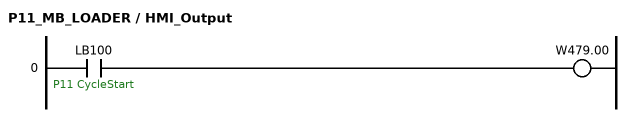
; [picture p120: P11_MB_LOADER / HMI_Output, rungs 0-0]
; rung 0
LD LB100  ; P11 CycleStart
OUT W479.00

### Section Autorun

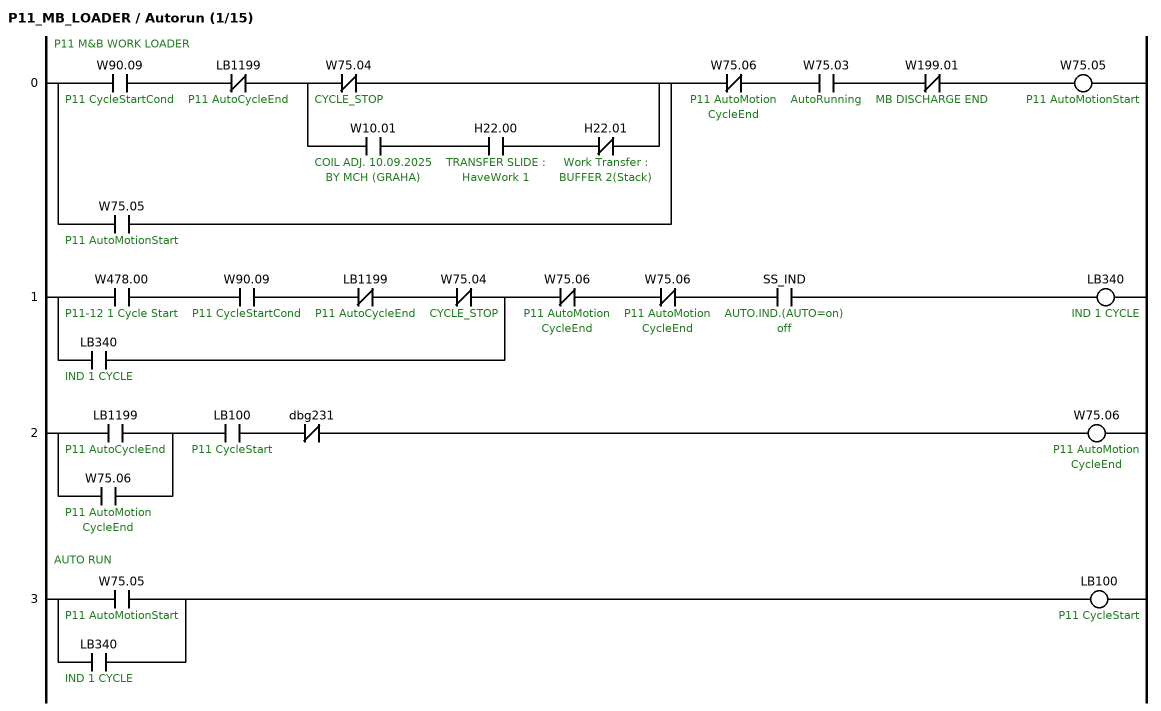
; rung 0: P11 M&B WORK LOADER
LD W90.09  ; P11 CycleStartCond
ANDNOT LB1199  ; P11 AutoCycleEnd
LDNOT W75.04  ; CYCLE_STOP
LD W10.01  ; COIL ADJ. 10.09.2025 BY MCH (GRAHA)
AND H22.00  ; TRANSFER SLIDE : HaveWork 1
ANDNOT H22.01  ; Work Transfer : BUFFER 2(Stack)
ORLD
ANDLD
OR W75.05  ; P11 AutoMotionStart
ANDNOT W75.06  ; P11 AutoMotion CycleEnd
AND W75.03  ; AutoRunning
ANDNOT W199.01  ; MB DISCHARGE END
OUT W75.05  ; P11 AutoMotionStart
; rung 1
LD W478.00  ; P11-12 1 Cycle Start
AND W90.09  ; P11 CycleStartCond
ANDNOT LB1199  ; P11 AutoCycleEnd
ANDNOT W75.04  ; CYCLE_STOP
OR LB340  ; IND 1 CYCLE
ANDNOT W75.06  ; P11 AutoMotion CycleEnd
ANDNOT W75.06  ; P11 AutoMotion CycleEnd
AND SS_IND  ; AUTO.IND.(AUTO=on) off
OUT LB340  ; IND 1 CYCLE
; rung 2
LD LB1199  ; P11 AutoCycleEnd
OR W75.06  ; P11 AutoMotion CycleEnd
AND LB100  ; P11 CycleStart
ANDNOT dbg231
OUT W75.06  ; P11 AutoMotion CycleEnd
; rung 3: AUTO RUN
LD W75.05  ; P11 AutoMotionStart
OR LB340  ; IND 1 CYCLE
OUT LB100  ; P11 CycleStart

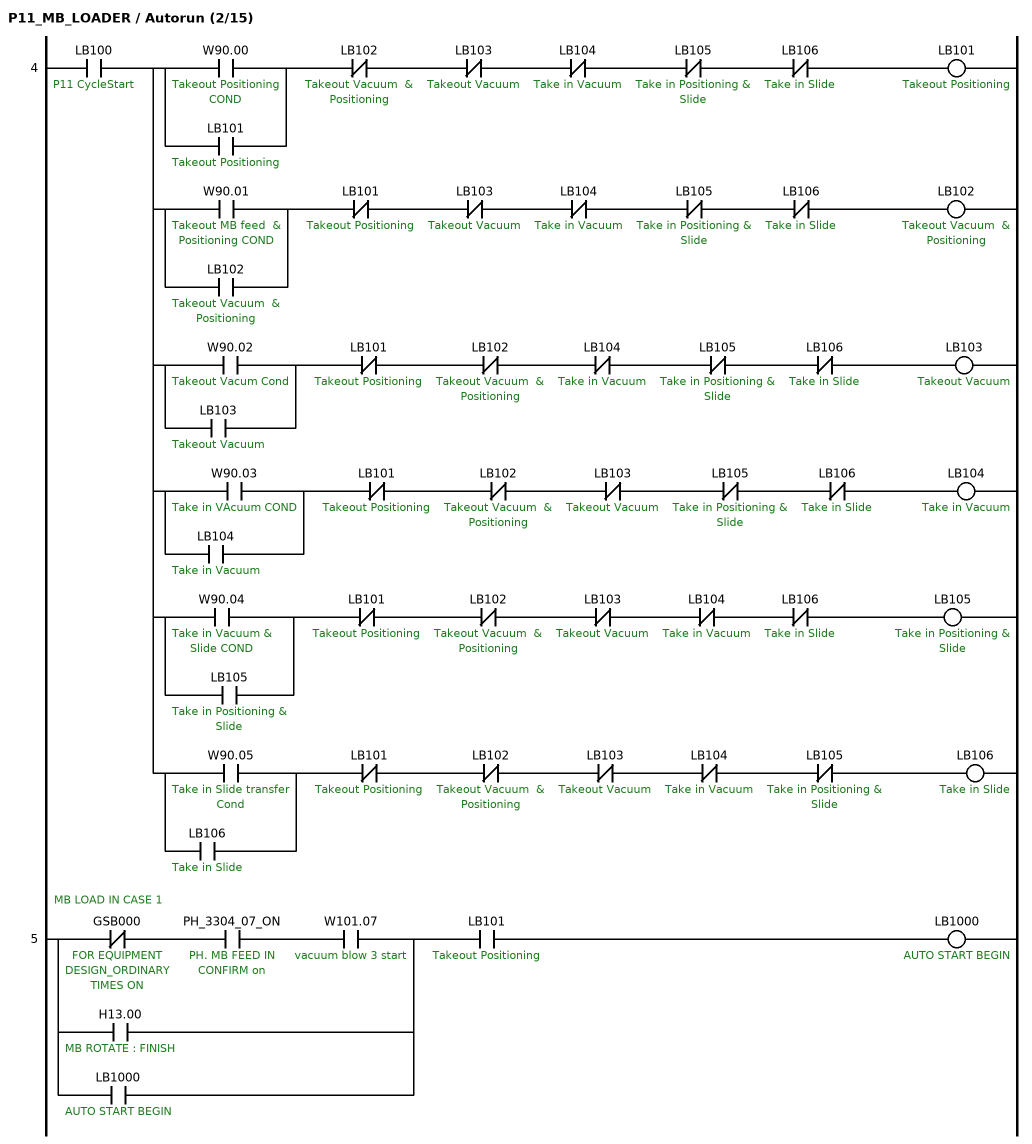
; rung 4
LD LB100  ; P11 CycleStart
OUT TR0
LD W90.00  ; Takeout Positioning COND
OR LB101  ; Takeout Positioning
ANDLD
ANDNOT LB102  ; Takeout Vacuum  & Positioning
ANDNOT LB103  ; Takeout Vacuum
ANDNOT LB104  ; Take in Vacuum
ANDNOT LB105  ; Take in Positioning & Slide
ANDNOT LB106  ; Take in Slide
OUT LB101  ; Takeout Positioning
LD TR0
LD W90.01  ; Takeout MB feed  & Positioning COND
OR LB102  ; Takeout Vacuum  & Positioning
ANDLD
ANDNOT LB101  ; Takeout Positioning
ANDNOT LB103  ; Takeout Vacuum
ANDNOT LB104  ; Take in Vacuum
ANDNOT LB105  ; Take in Positioning & Slide
ANDNOT LB106  ; Take in Slide
OUT LB102  ; Takeout Vacuum  & Positioning
LD TR0
LD W90.02  ; Takeout Vacum Cond
OR LB103  ; Takeout Vacuum
ANDLD
ANDNOT LB101  ; Takeout Positioning
ANDNOT LB102  ; Takeout Vacuum  & Positioning
ANDNOT LB104  ; Take in Vacuum
ANDNOT LB105  ; Take in Positioning & Slide
ANDNOT LB106  ; Take in Slide
OUT LB103  ; Takeout Vacuum
LD TR0
LD W90.03  ; Take in VAcuum COND
OR LB104  ; Take in Vacuum
ANDLD
ANDNOT LB101  ; Takeout Positioning
ANDNOT LB102  ; Takeout Vacuum  & Positioning
ANDNOT LB103  ; Takeout Vacuum
ANDNOT LB105  ; Take in Positioning & Slide
ANDNOT LB106  ; Take in Slide
OUT LB104  ; Take in Vacuum
LD TR0
LD W90.04  ; Take in Vacuum & Slide COND
OR LB105  ; Take in Positioning & Slide
ANDLD
ANDNOT LB101  ; Takeout Positioning
ANDNOT LB102  ; Takeout Vacuum  & Positioning
ANDNOT LB103  ; Takeout Vacuum
ANDNOT LB104  ; Take in Vacuum
ANDNOT LB106  ; Take in Slide
OUT LB105  ; Take in Positioning & Slide
LD TR0
LD W90.05  ; Take in Slide transfer Cond
OR LB106  ; Take in Slide
ANDLD
ANDNOT LB101  ; Takeout Positioning
ANDNOT LB102  ; Takeout Vacuum  & Positioning
ANDNOT LB103  ; Takeout Vacuum
ANDNOT LB104  ; Take in Vacuum
ANDNOT LB105  ; Take in Positioning & Slide
OUT LB106  ; Take in Slide
; rung 5: MB LOAD IN CASE 1
LDNOT GSB000  ; FOR EQUIPMENT DESIGN_ORDINARY TIMES ON
AND PH_3304_07_ON  ; PH. MB FEED IN CONFIRM on
AND W101.07  ; vacuum blow 3 start
OR H13.00  ; MB ROTATE : FINISH
OR LB1000  ; AUTO START BEGIN
AND LB101  ; Takeout Positioning
OUT LB1000  ; AUTO START BEGIN

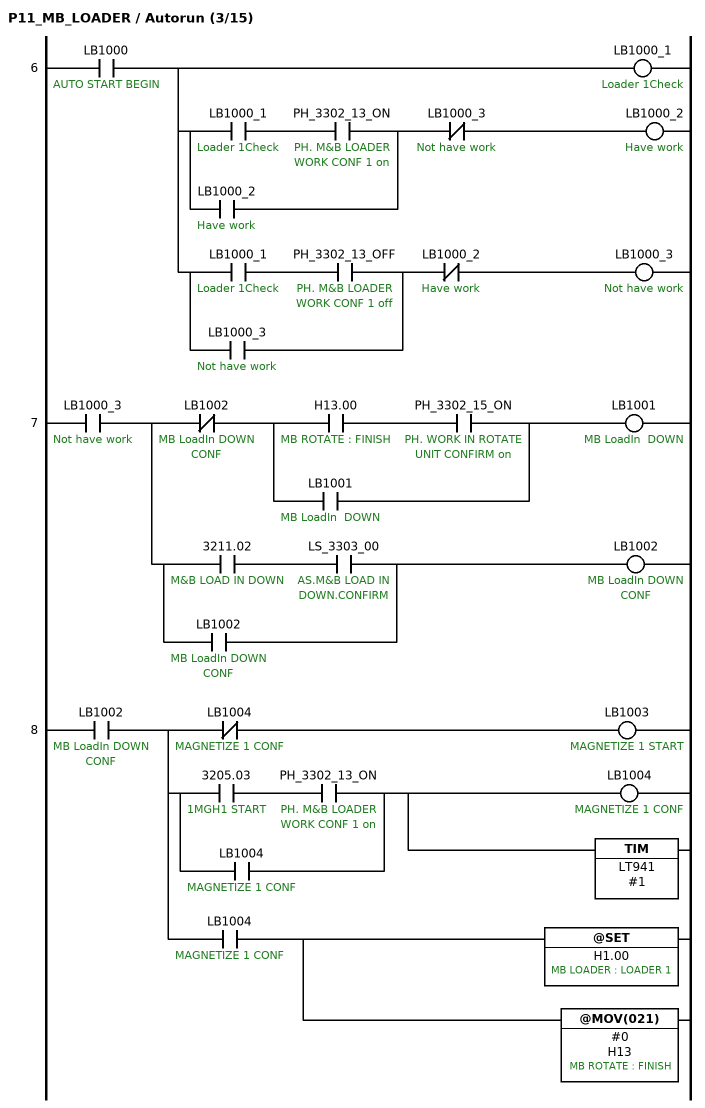
; rung 6
LD LB1000  ; AUTO START BEGIN
OUT TR0
OUT LB1000_1  ; Loader 1Check
LD LB1000_1  ; Loader 1Check
AND PH_3302_13_ON  ; PH. M&B LOADER WORK CONF 1 on
OR LB1000_2  ; Have work
ANDLD
ANDNOT LB1000_3  ; Not have work
OUT LB1000_2  ; Have work
LD TR0
LD LB1000_1  ; Loader 1Check
AND PH_3302_13_OFF  ; PH. M&B LOADER WORK CONF 1 off
OR LB1000_3  ; Not have work
ANDLD
ANDNOT LB1000_2  ; Have work
OUT LB1000_3  ; Not have work
; rung 7
LD LB1000_3  ; Not have work
OUT TR0
ANDNOT LB1002  ; MB LoadIn DOWN CONF
LD H13.00  ; MB ROTATE : FINISH
AND PH_3302_15_ON  ; PH. WORK IN ROTATE UNIT CONFIRM on
OR LB1001  ; MB LoadIn  DOWN
ANDLD
OUT LB1001  ; MB LoadIn  DOWN
LD TR0
LD 3211.02  ; M&B LOAD IN DOWN
AND LS_3303_00  ; AS.M&B LOAD IN DOWN.CONFIRM
OR LB1002  ; MB LoadIn DOWN CONF
ANDLD
OUT LB1002  ; MB LoadIn DOWN CONF
; rung 8
LD LB1002  ; MB LoadIn DOWN CONF
OUT TR0
ANDNOT LB1004  ; MAGNETIZE 1 CONF
OUT LB1003  ; MAGNETIZE 1 START
LD TR0
LD 3205.03  ; 1MGH1 START
AND PH_3302_13_ON  ; PH. M&B LOADER WORK CONF 1 on
OR LB1004  ; MAGNETIZE 1 CONF
ANDLD
OUT LB1004  ; MAGNETIZE 1 CONF
TIM LT941 #1
LD TR0
AND LB1004  ; MAGNETIZE 1 CONF
@SET H1.00  ; MB LOADER : LOADER 1
@MOV(021) #0 H13  ; MB ROTATE : FINISH

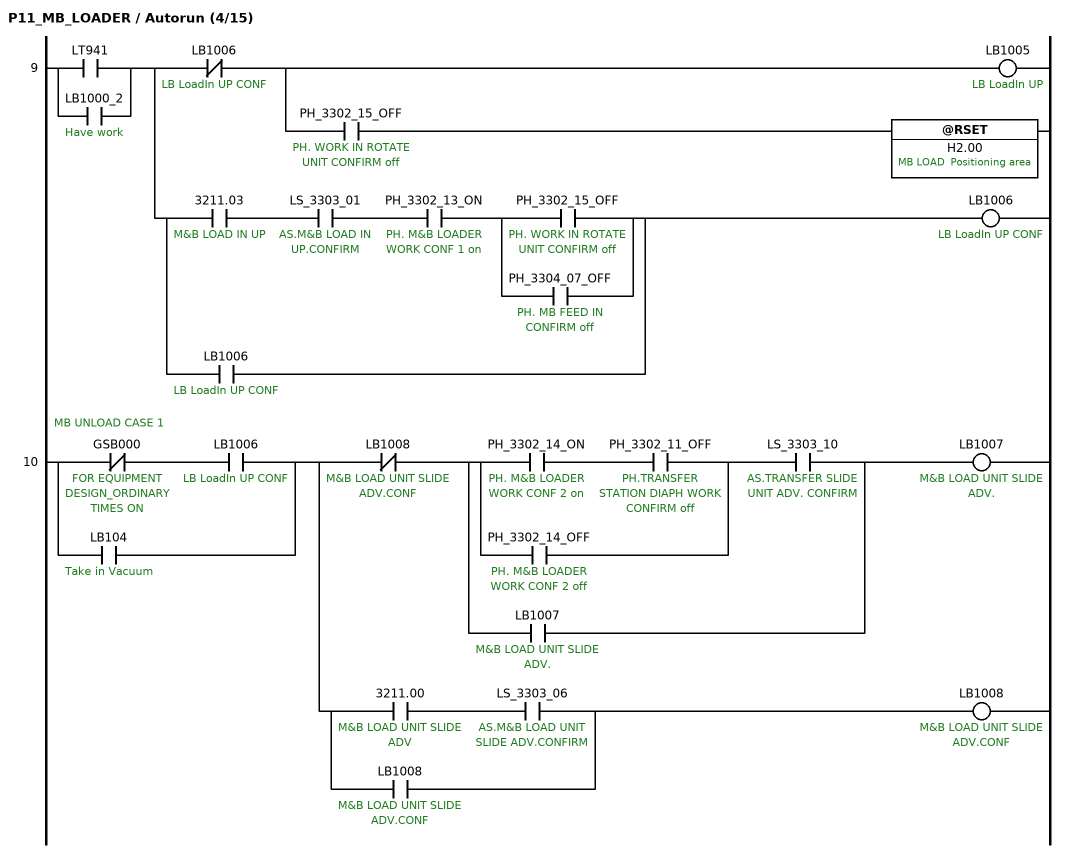
; rung 9
LD LT941
OR LB1000_2  ; Have work
OUT TR0
ANDNOT LB1006  ; LB LoadIn UP CONF
OUT LB1005  ; LB LoadIn UP
AND PH_3302_15_OFF  ; PH. WORK IN ROTATE UNIT CONFIRM off
@RSET H2.00  ; MB LOAD  Positioning area
LD TR0
LD 3211.03  ; M&B LOAD IN UP
AND LS_3303_01  ; AS.M&B LOAD IN UP.CONFIRM
AND PH_3302_13_ON  ; PH. M&B LOADER WORK CONF 1 on
LD PH_3302_15_OFF  ; PH. WORK IN ROTATE UNIT CONFIRM off
OR PH_3304_07_OFF  ; PH. MB FEED IN CONFIRM off
ANDLD
OR LB1006  ; LB LoadIn UP CONF
ANDLD
OUT LB1006  ; LB LoadIn UP CONF
; rung 10: MB UNLOAD CASE 1
LDNOT GSB000  ; FOR EQUIPMENT DESIGN_ORDINARY TIMES ON
AND LB1006  ; LB LoadIn UP CONF
OR LB104  ; Take in Vacuum
OUT TR0
ANDNOT LB1008  ; M&B LOAD UNIT SLIDE ADV.CONF
LD PH_3302_14_ON  ; PH. M&B LOADER WORK CONF 2 on
AND PH_3302_11_OFF  ; PH.TRANSFER STATION DIAPH WORK CONFIRM off
OR PH_3302_14_OFF  ; PH. M&B LOADER WORK CONF 2 off
AND LS_3303_10  ; AS.TRANSFER SLIDE UNIT ADV. CONFIRM
OR LB1007  ; M&B LOAD UNIT SLIDE ADV.
ANDLD
OUT LB1007  ; M&B LOAD UNIT SLIDE ADV.
LD TR0
LD 3211.00  ; M&B LOAD UNIT SLIDE ADV
AND LS_3303_06  ; AS.M&B LOAD UNIT SLIDE ADV.CONFIRM
OR LB1008  ; M&B LOAD UNIT SLIDE ADV.CONF
ANDLD
OUT LB1008  ; M&B LOAD UNIT SLIDE ADV.CONF

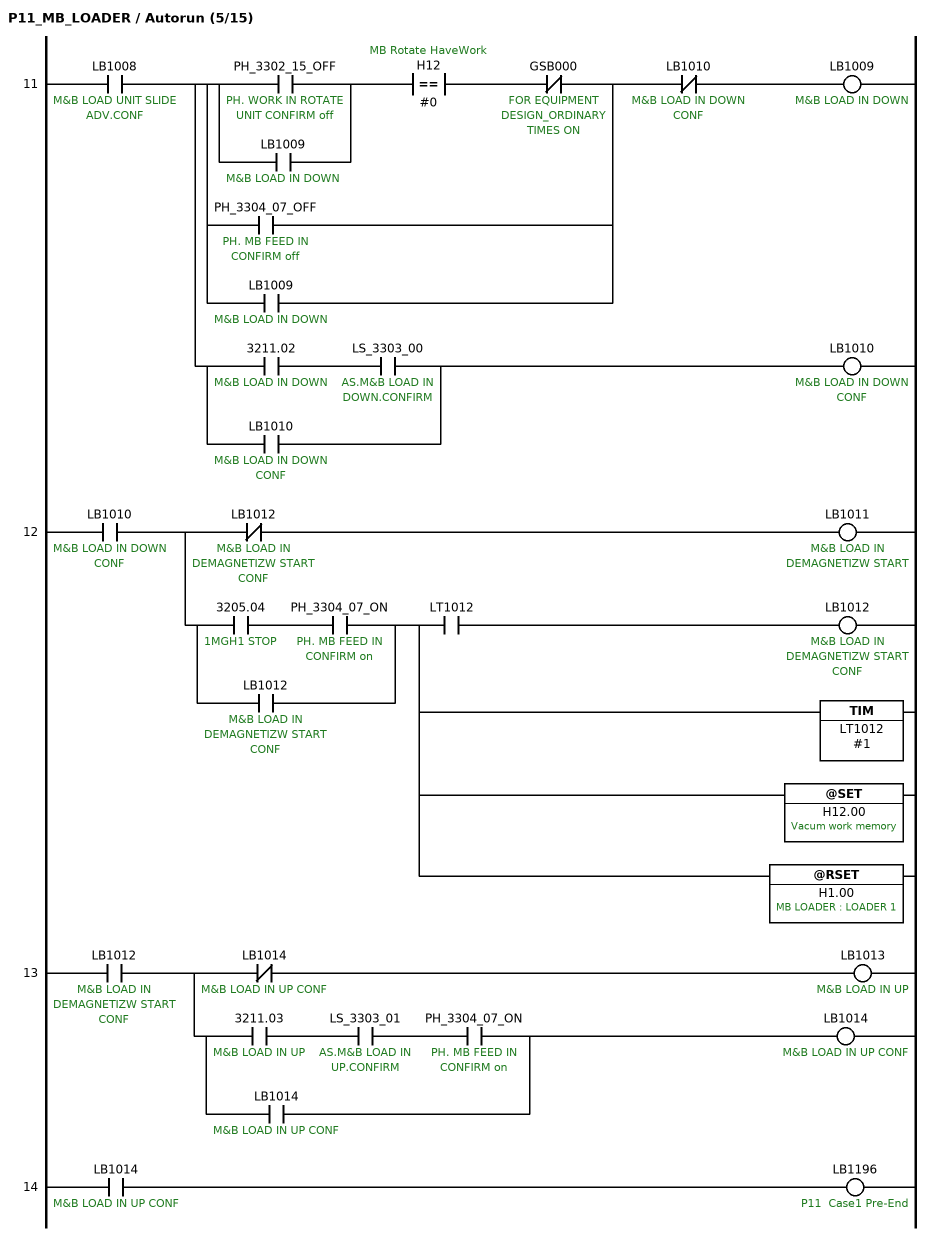
; rung 11
LD LB1008  ; M&B LOAD UNIT SLIDE ADV.CONF
OUT TR0
LD PH_3302_15_OFF  ; PH. WORK IN ROTATE UNIT CONFIRM off
OR LB1009  ; M&B LOAD IN DOWN
AND=(300) H12 #0  ; MB Rotate HaveWork
ANDNOT GSB000  ; FOR EQUIPMENT DESIGN_ORDINARY TIMES ON
LD PH_3304_07_OFF  ; PH. MB FEED IN CONFIRM off
OR LB1009  ; M&B LOAD IN DOWN
ORLD
ANDLD
ANDNOT LB1010  ; M&B LOAD IN DOWN CONF
OUT LB1009  ; M&B LOAD IN DOWN
LD TR0
LD 3211.02  ; M&B LOAD IN DOWN
AND LS_3303_00  ; AS.M&B LOAD IN DOWN.CONFIRM
OR LB1010  ; M&B LOAD IN DOWN CONF
ANDLD
OUT LB1010  ; M&B LOAD IN DOWN CONF
; rung 12
LD LB1010  ; M&B LOAD IN DOWN CONF
OUT TR0
ANDNOT LB1012  ; M&B LOAD IN DEMAGNETIZW START CONF
OUT LB1011  ; M&B LOAD IN DEMAGNETIZW START
LD TR0
LD 3205.04  ; 1MGH1 STOP
AND PH_3304_07_ON  ; PH. MB FEED IN CONFIRM on
OR LB1012  ; M&B LOAD IN DEMAGNETIZW START CONF
ANDLD
OUT TR0
AND LT1012
OUT LB1012  ; M&B LOAD IN DEMAGNETIZW START CONF
LD TR0
TIM LT1012 #1
@SET H12.00  ; Vacum work memory
@RSET H1.00  ; MB LOADER : LOADER 1
; rung 13
LD LB1012  ; M&B LOAD IN DEMAGNETIZW START CONF
OUT TR0
ANDNOT LB1014  ; M&B LOAD IN UP CONF
OUT LB1013  ; M&B LOAD IN UP
LD TR0
LD 3211.03  ; M&B LOAD IN UP
AND LS_3303_01  ; AS.M&B LOAD IN UP.CONFIRM
AND PH_3304_07_ON  ; PH. MB FEED IN CONFIRM on
OR LB1014  ; M&B LOAD IN UP CONF
ANDLD
OUT LB1014  ; M&B LOAD IN UP CONF
; rung 14
LD LB1014  ; M&B LOAD IN UP CONF
OUT LB1196  ; P11  Case1 Pre-End

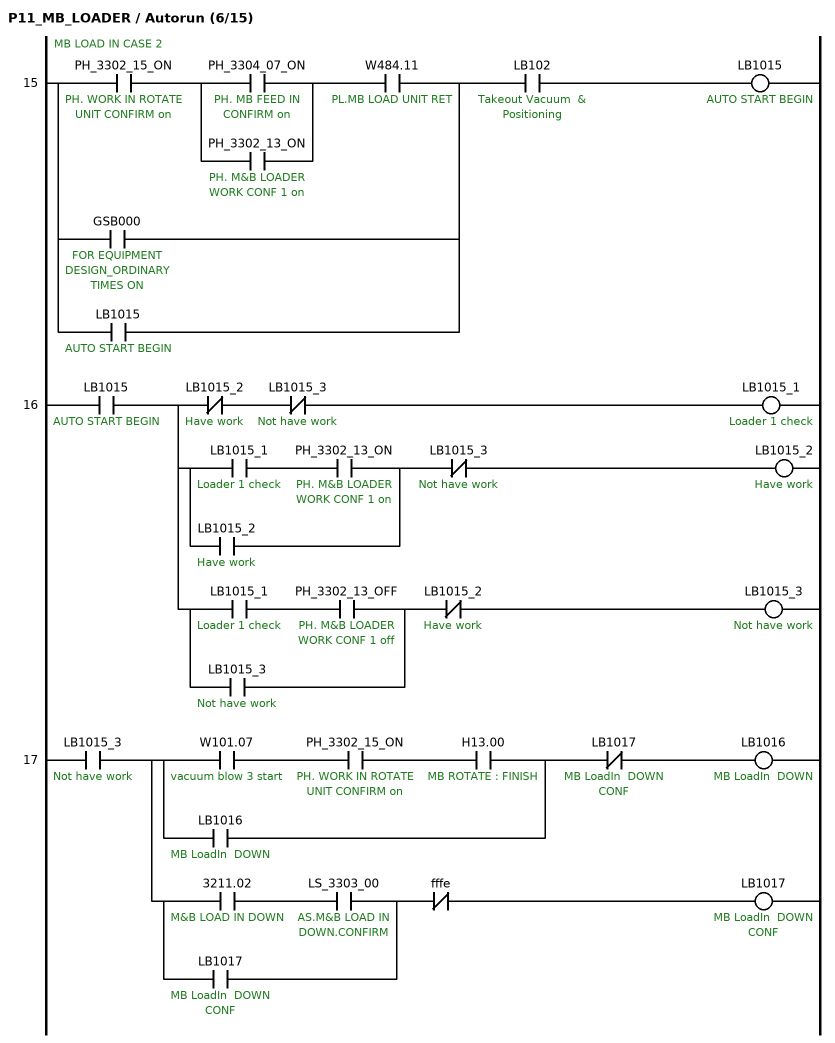
; rung 15: MB LOAD IN CASE 2
LD PH_3302_15_ON  ; PH. WORK IN ROTATE UNIT CONFIRM on
LD PH_3304_07_ON  ; PH. MB FEED IN CONFIRM on
OR PH_3302_13_ON  ; PH. M&B LOADER WORK CONF 1 on
ANDLD
AND W484.11  ; PL.MB LOAD UNIT RET
OR GSB000  ; FOR EQUIPMENT DESIGN_ORDINARY TIMES ON
OR LB1015  ; AUTO START BEGIN
AND LB102  ; Takeout Vacuum  & Positioning
OUT LB1015  ; AUTO START BEGIN
; rung 16
LD LB1015  ; AUTO START BEGIN
OUT TR0
ANDNOT LB1015_2  ; Have work
ANDNOT LB1015_3  ; Not have work
OUT LB1015_1  ; Loader 1 check
LD TR0
LD LB1015_1  ; Loader 1 check
AND PH_3302_13_ON  ; PH. M&B LOADER WORK CONF 1 on
OR LB1015_2  ; Have work
ANDLD
ANDNOT LB1015_3  ; Not have work
OUT LB1015_2  ; Have work
LD TR0
LD LB1015_1  ; Loader 1 check
AND PH_3302_13_OFF  ; PH. M&B LOADER WORK CONF 1 off
OR LB1015_3  ; Not have work
ANDLD
ANDNOT LB1015_2  ; Have work
OUT LB1015_3  ; Not have work
; rung 17
LD LB1015_3  ; Not have work
OUT TR0
LD W101.07  ; vacuum blow 3 start
AND PH_3302_15_ON  ; PH. WORK IN ROTATE UNIT CONFIRM on
AND H13.00  ; MB ROTATE : FINISH
OR LB1016  ; MB LoadIn  DOWN
ANDLD
ANDNOT LB1017  ; MB LoadIn  DOWN CONF
OUT LB1016  ; MB LoadIn  DOWN
LD TR0
LD 3211.02  ; M&B LOAD IN DOWN
AND LS_3303_00  ; AS.M&B LOAD IN DOWN.CONFIRM
OR LB1017  ; MB LoadIn  DOWN CONF
ANDLD
ANDNOT fffe
OUT LB1017  ; MB LoadIn  DOWN CONF

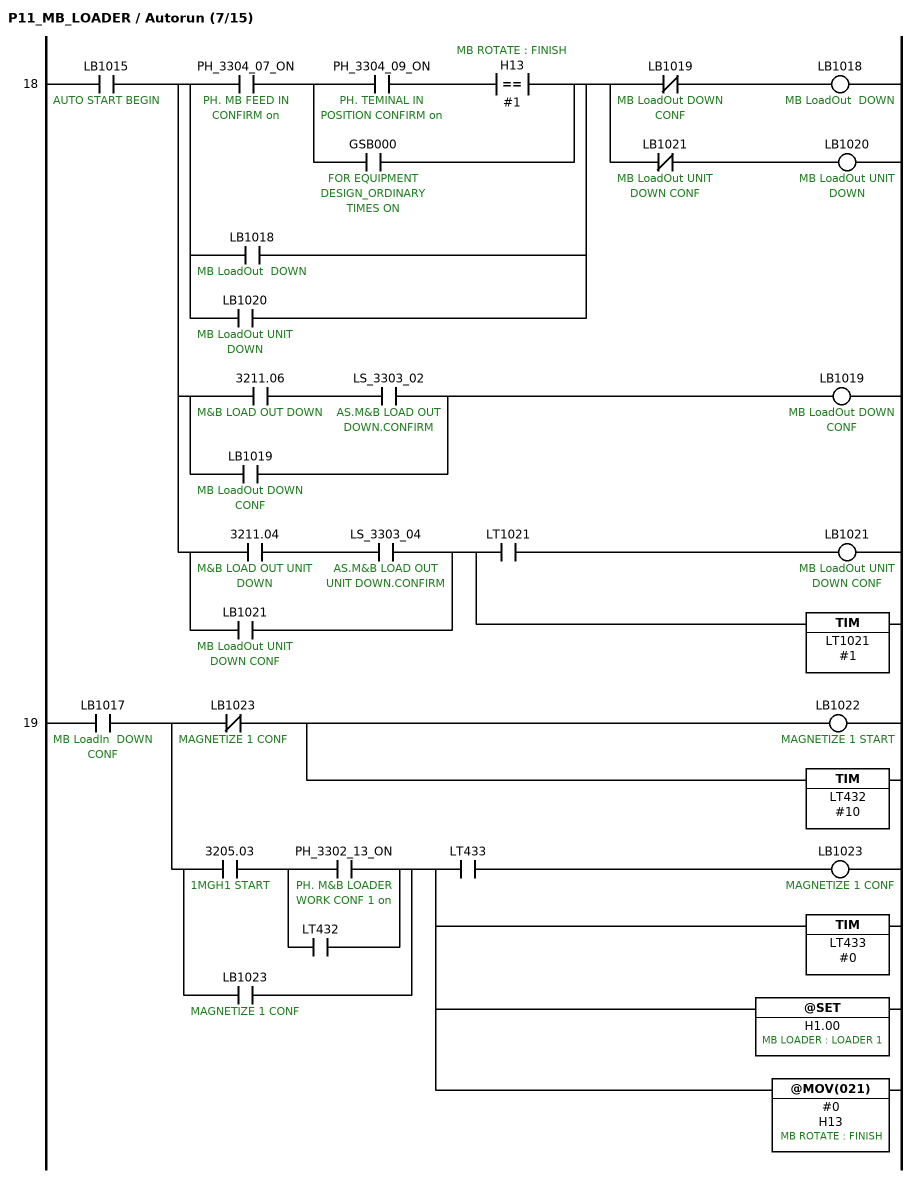
; rung 18
LD LB1015  ; AUTO START BEGIN
OUT TR0
LD PH_3304_07_ON  ; PH. MB FEED IN CONFIRM on
LD PH_3304_09_ON  ; PH. TEMINAL IN POSITION CONFIRM on
AND=(300) H13 #1  ; MB ROTATE : FINISH
OR GSB000  ; FOR EQUIPMENT DESIGN_ORDINARY TIMES ON
ANDLD
OR LB1018  ; MB LoadOut  DOWN
OR LB1020  ; MB LoadOut UNIT DOWN
ANDLD
OUT TR1
ANDNOT LB1019  ; MB LoadOut DOWN CONF
OUT LB1018  ; MB LoadOut  DOWN
LD TR1
ANDNOT LB1021  ; MB LoadOut UNIT DOWN CONF
OUT LB1020  ; MB LoadOut UNIT DOWN
LD TR0
LD 3211.06  ; M&B LOAD OUT DOWN
AND LS_3303_02  ; AS.M&B LOAD OUT DOWN.CONFIRM
OR LB1019  ; MB LoadOut DOWN CONF
ANDLD
OUT LB1019  ; MB LoadOut DOWN CONF
LD TR0
LD 3211.04  ; M&B LOAD OUT UNIT DOWN
AND LS_3303_04  ; AS.M&B LOAD OUT UNIT DOWN.CONFIRM
OR LB1021  ; MB LoadOut UNIT DOWN CONF
ANDLD
OUT TR0
AND LT1021
OUT LB1021  ; MB LoadOut UNIT DOWN CONF
LD TR0
TIM LT1021 #1
; rung 19
LD LB1017  ; MB LoadIn  DOWN CONF
OUT TR0
ANDNOT LB1023  ; MAGNETIZE 1 CONF
OUT LB1022  ; MAGNETIZE 1 START
TIM LT432 #10
LD TR0
LD 3205.03  ; 1MGH1 START
LD PH_3302_13_ON  ; PH. M&B LOADER WORK CONF 1 on
OR LT432
ANDLD
OR LB1023  ; MAGNETIZE 1 CONF
ANDLD
OUT TR0
AND LT433
OUT LB1023  ; MAGNETIZE 1 CONF
LD TR0
TIM LT433 #0
@SET H1.00  ; MB LOADER : LOADER 1
@MOV(021) #0 H13  ; MB ROTATE : FINISH

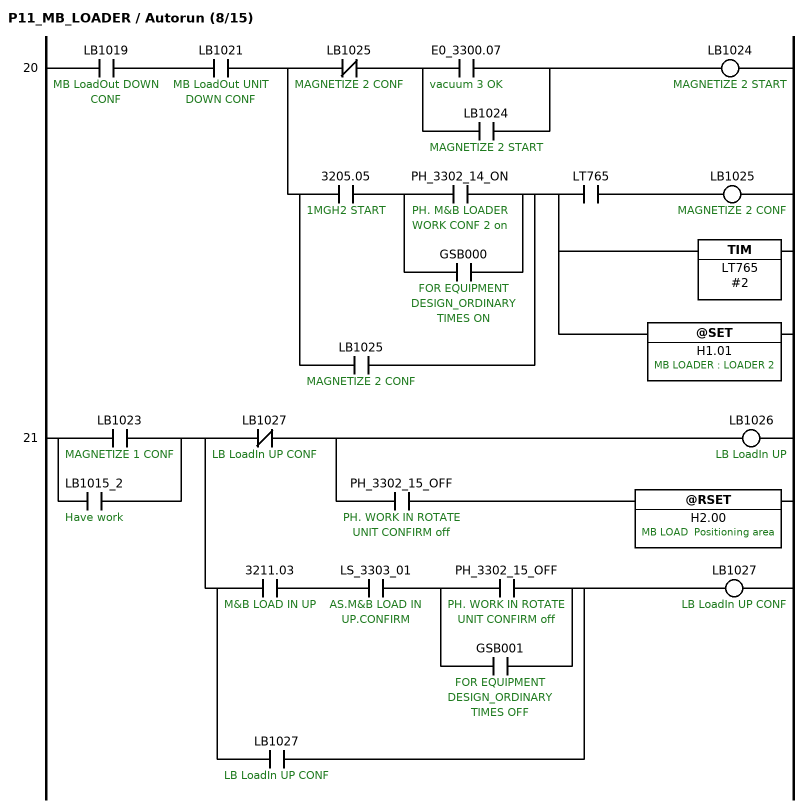
; rung 20
LD LB1019  ; MB LoadOut DOWN CONF
AND LB1021  ; MB LoadOut UNIT DOWN CONF
OUT TR0
ANDNOT LB1025  ; MAGNETIZE 2 CONF
LD E0_3300.07  ; vacuum 3 OK
OR LB1024  ; MAGNETIZE 2 START
ANDLD
OUT LB1024  ; MAGNETIZE 2 START
LD TR0
LD 3205.05  ; 1MGH2 START
LD PH_3302_14_ON  ; PH. M&B LOADER WORK CONF 2 on
OR GSB000  ; FOR EQUIPMENT DESIGN_ORDINARY TIMES ON
ANDLD
OR LB1025  ; MAGNETIZE 2 CONF
ANDLD
OUT TR0
AND LT765
OUT LB1025  ; MAGNETIZE 2 CONF
LD TR0
TIM LT765 #2
@SET H1.01  ; MB LOADER : LOADER 2
; rung 21
LD LB1023  ; MAGNETIZE 1 CONF
OR LB1015_2  ; Have work
OUT TR0
ANDNOT LB1027  ; LB LoadIn UP CONF
OUT LB1026  ; LB LoadIn UP
AND PH_3302_15_OFF  ; PH. WORK IN ROTATE UNIT CONFIRM off
@RSET H2.00  ; MB LOAD  Positioning area
LD TR0
LD 3211.03  ; M&B LOAD IN UP
AND LS_3303_01  ; AS.M&B LOAD IN UP.CONFIRM
LD PH_3302_15_OFF  ; PH. WORK IN ROTATE UNIT CONFIRM off
OR GSB001  ; FOR EQUIPMENT DESIGN_ORDINARY TIMES OFF
ANDLD
OR LB1027  ; LB LoadIn UP CONF
ANDLD
OUT LB1027  ; LB LoadIn UP CONF

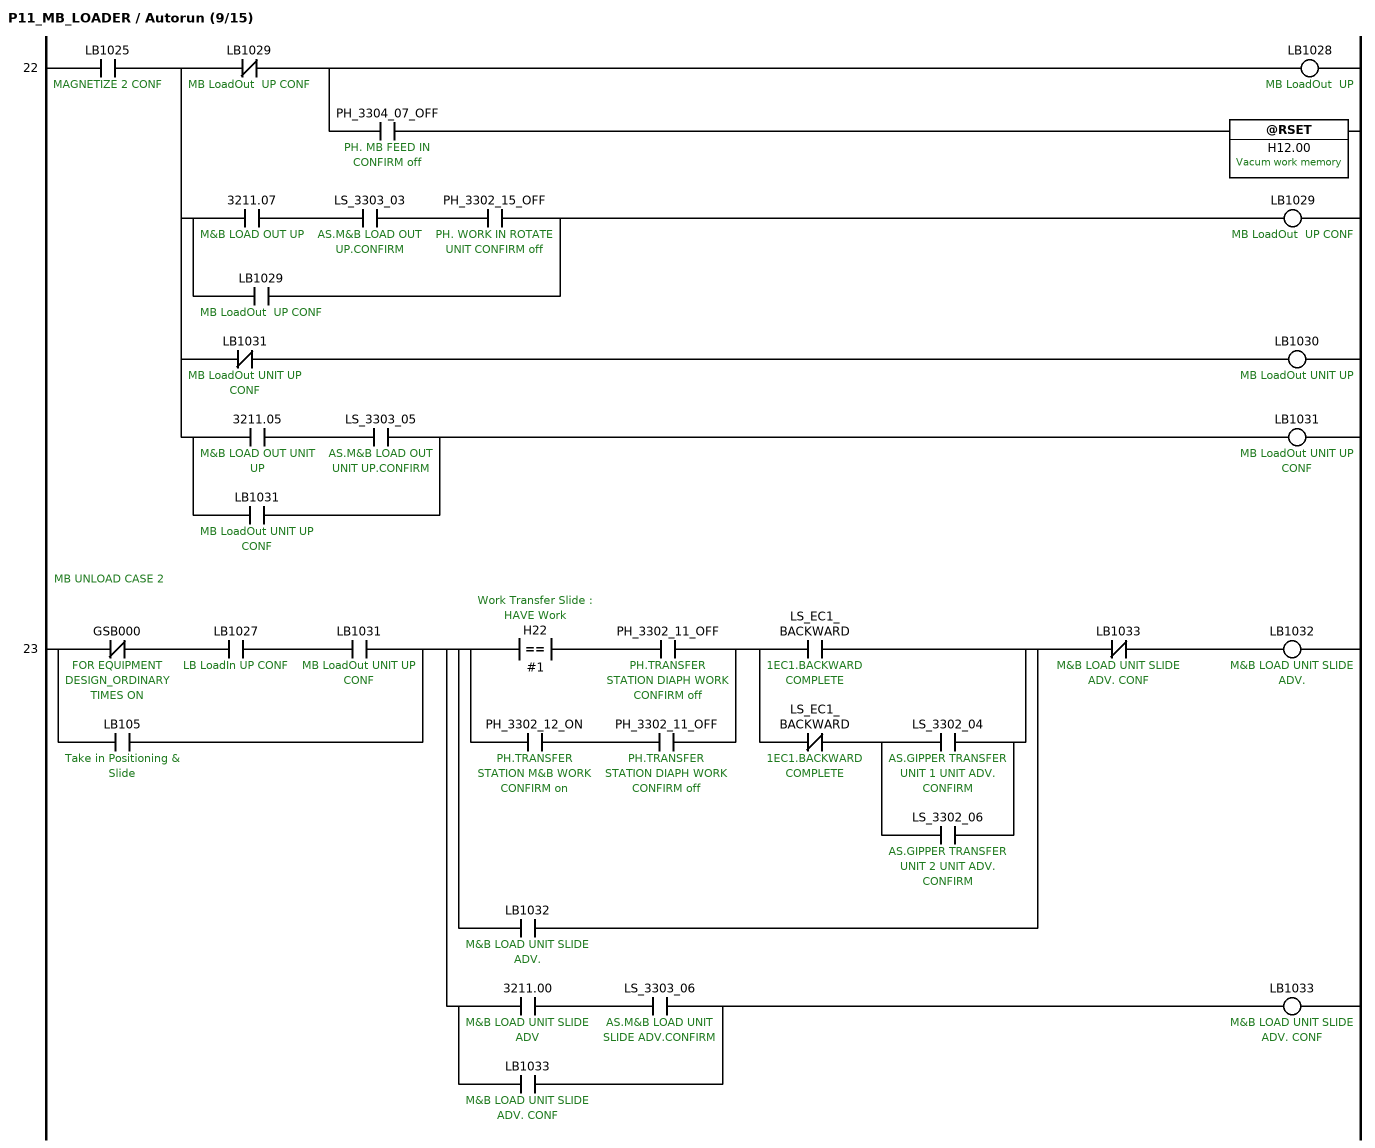
; rung 22
LD LB1025  ; MAGNETIZE 2 CONF
OUT TR0
ANDNOT LB1029  ; MB LoadOut  UP CONF
OUT LB1028  ; MB LoadOut  UP
AND PH_3304_07_OFF  ; PH. MB FEED IN CONFIRM off
@RSET H12.00  ; Vacum work memory
LD TR0
LD 3211.07  ; M&B LOAD OUT UP
AND LS_3303_03  ; AS.M&B LOAD OUT UP.CONFIRM
AND PH_3302_15_OFF  ; PH. WORK IN ROTATE UNIT CONFIRM off
OR LB1029  ; MB LoadOut  UP CONF
ANDLD
OUT LB1029  ; MB LoadOut  UP CONF
LD TR0
ANDNOT LB1031  ; MB LoadOut UNIT UP CONF
OUT LB1030  ; MB LoadOut UNIT UP
LD TR0
LD 3211.05  ; M&B LOAD OUT UNIT UP
AND LS_3303_05  ; AS.M&B LOAD OUT UNIT UP.CONFIRM
OR LB1031  ; MB LoadOut UNIT UP CONF
ANDLD
OUT LB1031  ; MB LoadOut UNIT UP CONF
; rung 23: MB UNLOAD CASE 2
LDNOT GSB000  ; FOR EQUIPMENT DESIGN_ORDINARY TIMES ON
AND LB1027  ; LB LoadIn UP CONF
AND LB1031  ; MB LoadOut UNIT UP CONF
OR LB105  ; Take in Positioning & Slide
OUT TR0
LD=(300) H22 #1  ; Work Transfer Slide : HAVE Work
AND PH_3302_11_OFF  ; PH.TRANSFER STATION DIAPH WORK CONFIRM off
LD PH_3302_12_ON  ; PH.TRANSFER STATION M&B WORK CONFIRM on
AND PH_3302_11_OFF  ; PH.TRANSFER STATION DIAPH WORK CONFIRM off
ORLD
LD LS_EC1_BACKWARD  ; 1EC1.BACKWARD COMPLETE
LDNOT LS_EC1_BACKWARD  ; 1EC1.BACKWARD COMPLETE
LD LS_3302_04  ; AS.GIPPER TRANSFER UNIT 1 UNIT ADV. CONFIRM
OR LS_3302_06  ; AS.GIPPER TRANSFER UNIT 2 UNIT ADV. CONFIRM
ANDLD
ORLD
ANDLD
OR LB1032  ; M&B LOAD UNIT SLIDE ADV.
ANDLD
ANDNOT LB1033  ; M&B LOAD UNIT SLIDE ADV. CONF
OUT LB1032  ; M&B LOAD UNIT SLIDE ADV.
LD TR0
LD 3211.00  ; M&B LOAD UNIT SLIDE ADV
AND LS_3303_06  ; AS.M&B LOAD UNIT SLIDE ADV.CONFIRM
OR LB1033  ; M&B LOAD UNIT SLIDE ADV. CONF
ANDLD
OUT LB1033  ; M&B LOAD UNIT SLIDE ADV. CONF

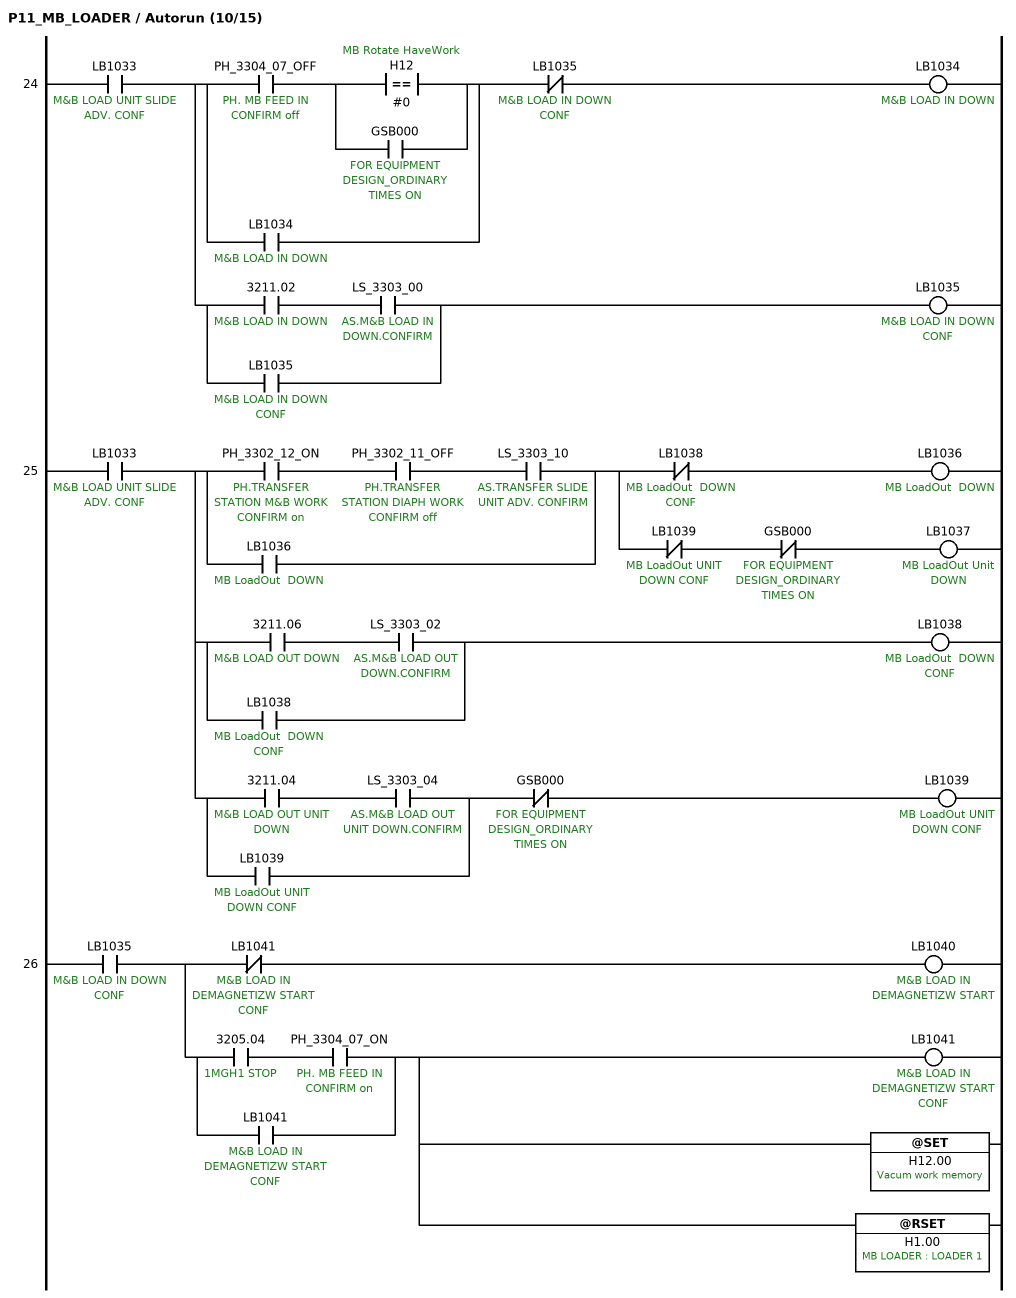
; rung 24
LD LB1033  ; M&B LOAD UNIT SLIDE ADV. CONF
OUT TR0
LD PH_3304_07_OFF  ; PH. MB FEED IN CONFIRM off
LD=(300) H12 #0  ; MB Rotate HaveWork
OR GSB000  ; FOR EQUIPMENT DESIGN_ORDINARY TIMES ON
ANDLD
OR LB1034  ; M&B LOAD IN DOWN
ANDLD
ANDNOT LB1035  ; M&B LOAD IN DOWN CONF
OUT LB1034  ; M&B LOAD IN DOWN
LD TR0
LD 3211.02  ; M&B LOAD IN DOWN
AND LS_3303_00  ; AS.M&B LOAD IN DOWN.CONFIRM
OR LB1035  ; M&B LOAD IN DOWN CONF
ANDLD
OUT LB1035  ; M&B LOAD IN DOWN CONF
; rung 25
LD LB1033  ; M&B LOAD UNIT SLIDE ADV. CONF
OUT TR0
LD PH_3302_12_ON  ; PH.TRANSFER STATION M&B WORK CONFIRM on
AND PH_3302_11_OFF  ; PH.TRANSFER STATION DIAPH WORK CONFIRM off
AND LS_3303_10  ; AS.TRANSFER SLIDE UNIT ADV. CONFIRM
OR LB1036  ; MB LoadOut  DOWN
ANDLD
OUT TR1
ANDNOT LB1038  ; MB LoadOut  DOWN CONF
OUT LB1036  ; MB LoadOut  DOWN
LD TR1
ANDNOT LB1039  ; MB LoadOut UNIT DOWN CONF
ANDNOT GSB000  ; FOR EQUIPMENT DESIGN_ORDINARY TIMES ON
OUT LB1037  ; MB LoadOut Unit  DOWN
LD TR0
LD 3211.06  ; M&B LOAD OUT DOWN
AND LS_3303_02  ; AS.M&B LOAD OUT DOWN.CONFIRM
OR LB1038  ; MB LoadOut  DOWN CONF
ANDLD
OUT LB1038  ; MB LoadOut  DOWN CONF
LD TR0
LD 3211.04  ; M&B LOAD OUT UNIT DOWN
AND LS_3303_04  ; AS.M&B LOAD OUT UNIT DOWN.CONFIRM
OR LB1039  ; MB LoadOut UNIT DOWN CONF
ANDLD
ANDNOT GSB000  ; FOR EQUIPMENT DESIGN_ORDINARY TIMES ON
OUT LB1039  ; MB LoadOut UNIT DOWN CONF
; rung 26
LD LB1035  ; M&B LOAD IN DOWN CONF
OUT TR0
ANDNOT LB1041  ; M&B LOAD IN DEMAGNETIZW START CONF
OUT LB1040  ; M&B LOAD IN DEMAGNETIZW START
LD TR0
LD 3205.04  ; 1MGH1 STOP
AND PH_3304_07_ON  ; PH. MB FEED IN CONFIRM on
OR LB1041  ; M&B LOAD IN DEMAGNETIZW START CONF
ANDLD
OUT LB1041  ; M&B LOAD IN DEMAGNETIZW START CONF
@SET H12.00  ; Vacum work memory
@RSET H1.00  ; MB LOADER : LOADER 1

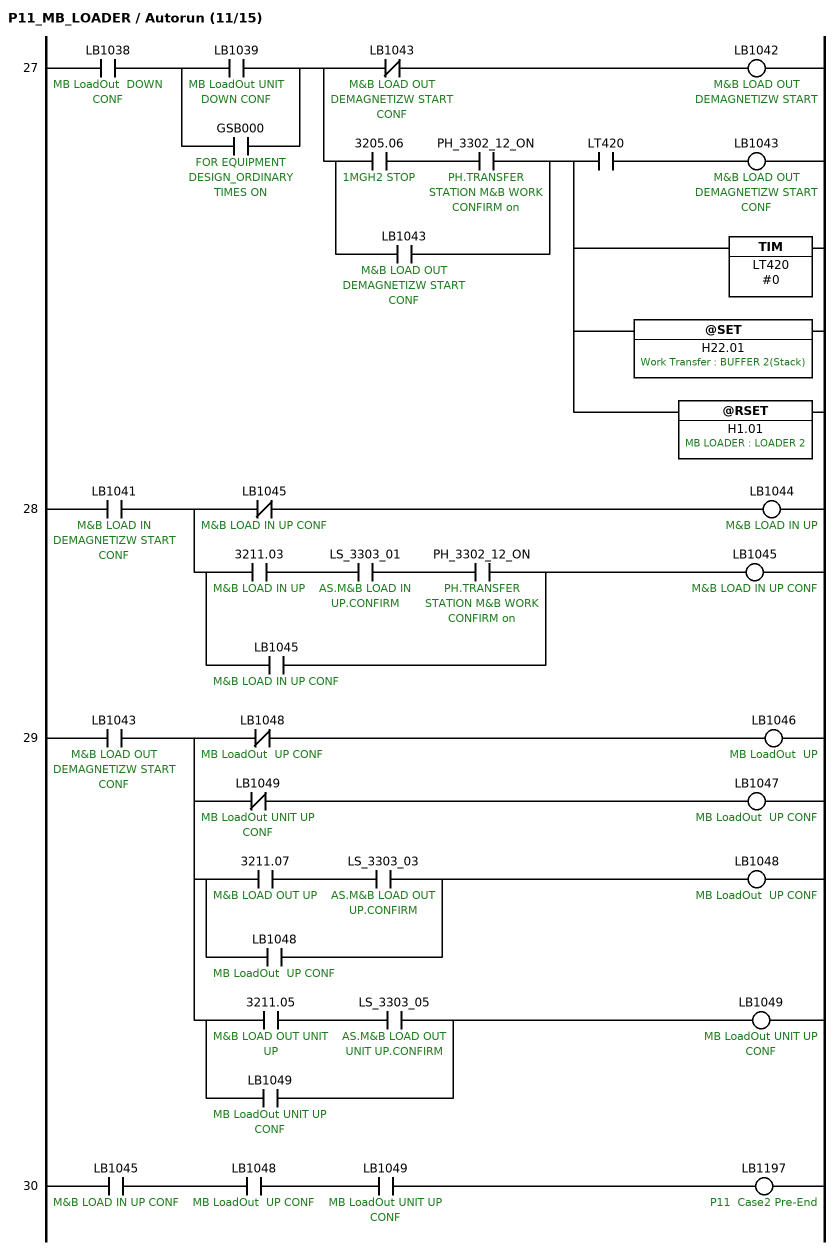
; rung 27
LD LB1038  ; MB LoadOut  DOWN CONF
LD LB1039  ; MB LoadOut UNIT DOWN CONF
OR GSB000  ; FOR EQUIPMENT DESIGN_ORDINARY TIMES ON
ANDLD
OUT TR0
ANDNOT LB1043  ; M&B LOAD OUT DEMAGNETIZW START CONF
OUT LB1042  ; M&B LOAD OUT DEMAGNETIZW START
LD TR0
LD 3205.06  ; 1MGH2 STOP
AND PH_3302_12_ON  ; PH.TRANSFER STATION M&B WORK CONFIRM on
OR LB1043  ; M&B LOAD OUT DEMAGNETIZW START CONF
ANDLD
OUT TR0
AND LT420
OUT LB1043  ; M&B LOAD OUT DEMAGNETIZW START CONF
LD TR0
TIM LT420 #0
@SET H22.01  ; Work Transfer : BUFFER 2(Stack)
@RSET H1.01  ; MB LOADER : LOADER 2
; rung 28
LD LB1041  ; M&B LOAD IN DEMAGNETIZW START CONF
OUT TR0
ANDNOT LB1045  ; M&B LOAD IN UP CONF
OUT LB1044  ; M&B LOAD IN UP
LD TR0
LD 3211.03  ; M&B LOAD IN UP
AND LS_3303_01  ; AS.M&B LOAD IN UP.CONFIRM
AND PH_3302_12_ON  ; PH.TRANSFER STATION M&B WORK CONFIRM on
OR LB1045  ; M&B LOAD IN UP CONF
ANDLD
OUT LB1045  ; M&B LOAD IN UP CONF
; rung 29
LD LB1043  ; M&B LOAD OUT DEMAGNETIZW START CONF
OUT TR0
ANDNOT LB1048  ; MB LoadOut  UP CONF
OUT LB1046  ; MB LoadOut  UP
LD TR0
ANDNOT LB1049  ; MB LoadOut UNIT UP CONF
OUT LB1047  ; MB LoadOut  UP CONF
LD TR0
LD 3211.07  ; M&B LOAD OUT UP
AND LS_3303_03  ; AS.M&B LOAD OUT UP.CONFIRM
OR LB1048  ; MB LoadOut  UP CONF
ANDLD
OUT LB1048  ; MB LoadOut  UP CONF
LD TR0
LD 3211.05  ; M&B LOAD OUT UNIT UP
AND LS_3303_05  ; AS.M&B LOAD OUT UNIT UP.CONFIRM
OR LB1049  ; MB LoadOut UNIT UP CONF
ANDLD
OUT LB1049  ; MB LoadOut UNIT UP CONF
; rung 30
LD LB1045  ; M&B LOAD IN UP CONF
AND LB1048  ; MB LoadOut  UP CONF
AND LB1049  ; MB LoadOut UNIT UP CONF
OUT LB1197  ; P11  Case2 Pre-End

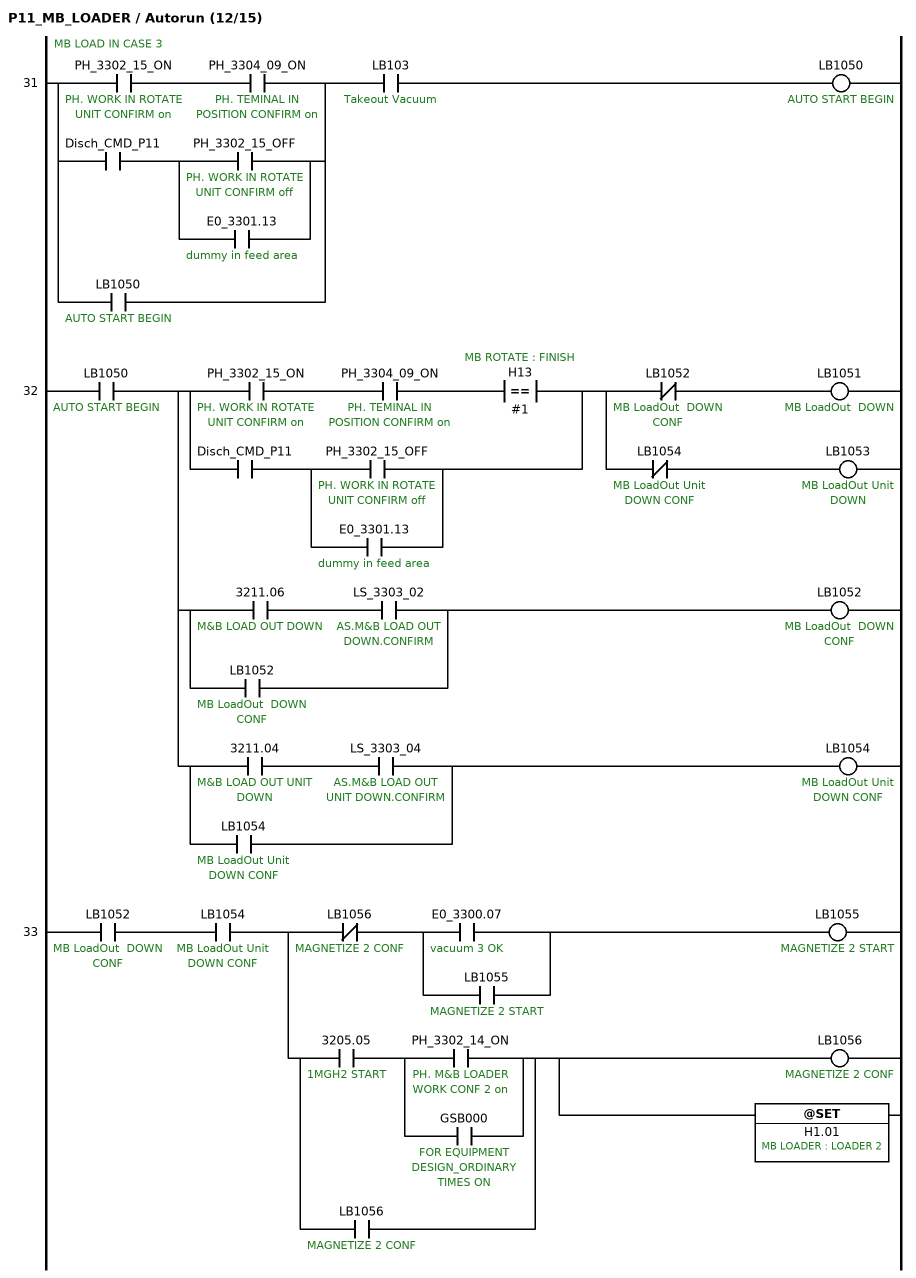
; rung 31: MB LOAD IN CASE 3
LD PH_3302_15_ON  ; PH. WORK IN ROTATE UNIT CONFIRM on
AND PH_3304_09_ON  ; PH. TEMINAL IN POSITION CONFIRM on
LD Disch_CMD_P11
LD PH_3302_15_OFF  ; PH. WORK IN ROTATE UNIT CONFIRM off
OR E0_3301.13  ; dummy in feed area
ANDLD
ORLD
OR LB1050  ; AUTO START BEGIN
AND LB103  ; Takeout Vacuum
OUT LB1050  ; AUTO START BEGIN
; rung 32
LD LB1050  ; AUTO START BEGIN
OUT TR0
LD PH_3302_15_ON  ; PH. WORK IN ROTATE UNIT CONFIRM on
AND PH_3304_09_ON  ; PH. TEMINAL IN POSITION CONFIRM on
AND=(300) H13 #1  ; MB ROTATE : FINISH
LD Disch_CMD_P11
LD PH_3302_15_OFF  ; PH. WORK IN ROTATE UNIT CONFIRM off
OR E0_3301.13  ; dummy in feed area
ANDLD
ORLD
ANDLD
OUT TR1
ANDNOT LB1052  ; MB LoadOut  DOWN CONF
OUT LB1051  ; MB LoadOut  DOWN
LD TR1
ANDNOT LB1054  ; MB LoadOut Unit DOWN CONF
OUT LB1053  ; MB LoadOut Unit DOWN
LD TR0
LD 3211.06  ; M&B LOAD OUT DOWN
AND LS_3303_02  ; AS.M&B LOAD OUT DOWN.CONFIRM
OR LB1052  ; MB LoadOut  DOWN CONF
ANDLD
OUT LB1052  ; MB LoadOut  DOWN CONF
LD TR0
LD 3211.04  ; M&B LOAD OUT UNIT DOWN
AND LS_3303_04  ; AS.M&B LOAD OUT UNIT DOWN.CONFIRM
OR LB1054  ; MB LoadOut Unit DOWN CONF
ANDLD
OUT LB1054  ; MB LoadOut Unit DOWN CONF
; rung 33
LD LB1052  ; MB LoadOut  DOWN CONF
AND LB1054  ; MB LoadOut Unit DOWN CONF
OUT TR0
ANDNOT LB1056  ; MAGNETIZE 2 CONF
LD E0_3300.07  ; vacuum 3 OK
OR LB1055  ; MAGNETIZE 2 START
ANDLD
OUT LB1055  ; MAGNETIZE 2 START
LD TR0
LD 3205.05  ; 1MGH2 START
LD PH_3302_14_ON  ; PH. M&B LOADER WORK CONF 2 on
OR GSB000  ; FOR EQUIPMENT DESIGN_ORDINARY TIMES ON
ANDLD
OR LB1056  ; MAGNETIZE 2 CONF
ANDLD
OUT LB1056  ; MAGNETIZE 2 CONF
@SET H1.01  ; MB LOADER : LOADER 2

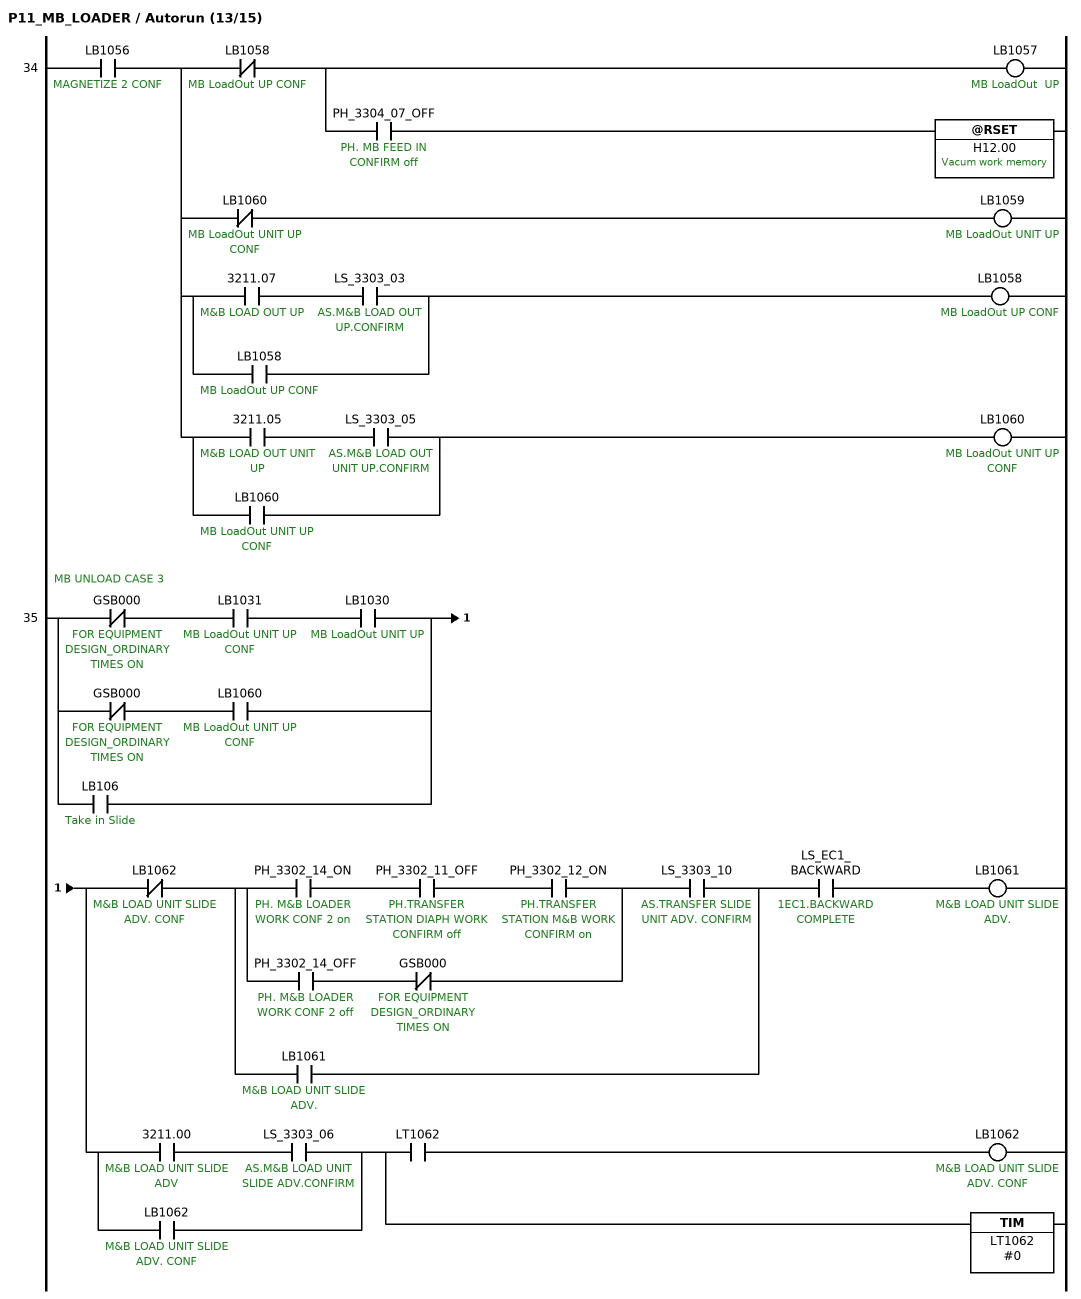
; rung 34
LD LB1056  ; MAGNETIZE 2 CONF
OUT TR0
ANDNOT LB1058  ; MB LoadOut UP CONF
OUT LB1057  ; MB LoadOut  UP
AND PH_3304_07_OFF  ; PH. MB FEED IN CONFIRM off
@RSET H12.00  ; Vacum work memory
LD TR0
ANDNOT LB1060  ; MB LoadOut UNIT UP CONF
OUT LB1059  ; MB LoadOut UNIT UP
LD TR0
LD 3211.07  ; M&B LOAD OUT UP
AND LS_3303_03  ; AS.M&B LOAD OUT UP.CONFIRM
OR LB1058  ; MB LoadOut UP CONF
ANDLD
OUT LB1058  ; MB LoadOut UP CONF
LD TR0
LD 3211.05  ; M&B LOAD OUT UNIT UP
AND LS_3303_05  ; AS.M&B LOAD OUT UNIT UP.CONFIRM
OR LB1060  ; MB LoadOut UNIT UP CONF
ANDLD
OUT LB1060  ; MB LoadOut UNIT UP CONF
; rung 35: MB UNLOAD CASE 3
LDNOT GSB000  ; FOR EQUIPMENT DESIGN_ORDINARY TIMES ON
AND LB1031  ; MB LoadOut UNIT UP CONF
AND LB1030  ; MB LoadOut UNIT UP
LDNOT GSB000  ; FOR EQUIPMENT DESIGN_ORDINARY TIMES ON
AND LB1060  ; MB LoadOut UNIT UP CONF
ORLD
OR LB106  ; Take in Slide
OUT TR0
ANDNOT LB1062  ; M&B LOAD UNIT SLIDE ADV. CONF
LD PH_3302_14_ON  ; PH. M&B LOADER WORK CONF 2 on
AND PH_3302_11_OFF  ; PH.TRANSFER STATION DIAPH WORK CONFIRM off
AND PH_3302_12_ON  ; PH.TRANSFER STATION M&B WORK CONFIRM on
LD PH_3302_14_OFF  ; PH. M&B LOADER WORK CONF 2 off
ANDNOT GSB000  ; FOR EQUIPMENT DESIGN_ORDINARY TIMES ON
ORLD
AND LS_3303_10  ; AS.TRANSFER SLIDE UNIT ADV. CONFIRM
OR LB1061  ; M&B LOAD UNIT SLIDE ADV.
ANDLD
AND LS_EC1_BACKWARD  ; 1EC1.BACKWARD COMPLETE
OUT LB1061  ; M&B LOAD UNIT SLIDE ADV.
LD TR0
LD 3211.00  ; M&B LOAD UNIT SLIDE ADV
AND LS_3303_06  ; AS.M&B LOAD UNIT SLIDE ADV.CONFIRM
OR LB1062  ; M&B LOAD UNIT SLIDE ADV. CONF
ANDLD
OUT TR0
AND LT1062
OUT LB1062  ; M&B LOAD UNIT SLIDE ADV. CONF
LD TR0
TIM LT1062 #0

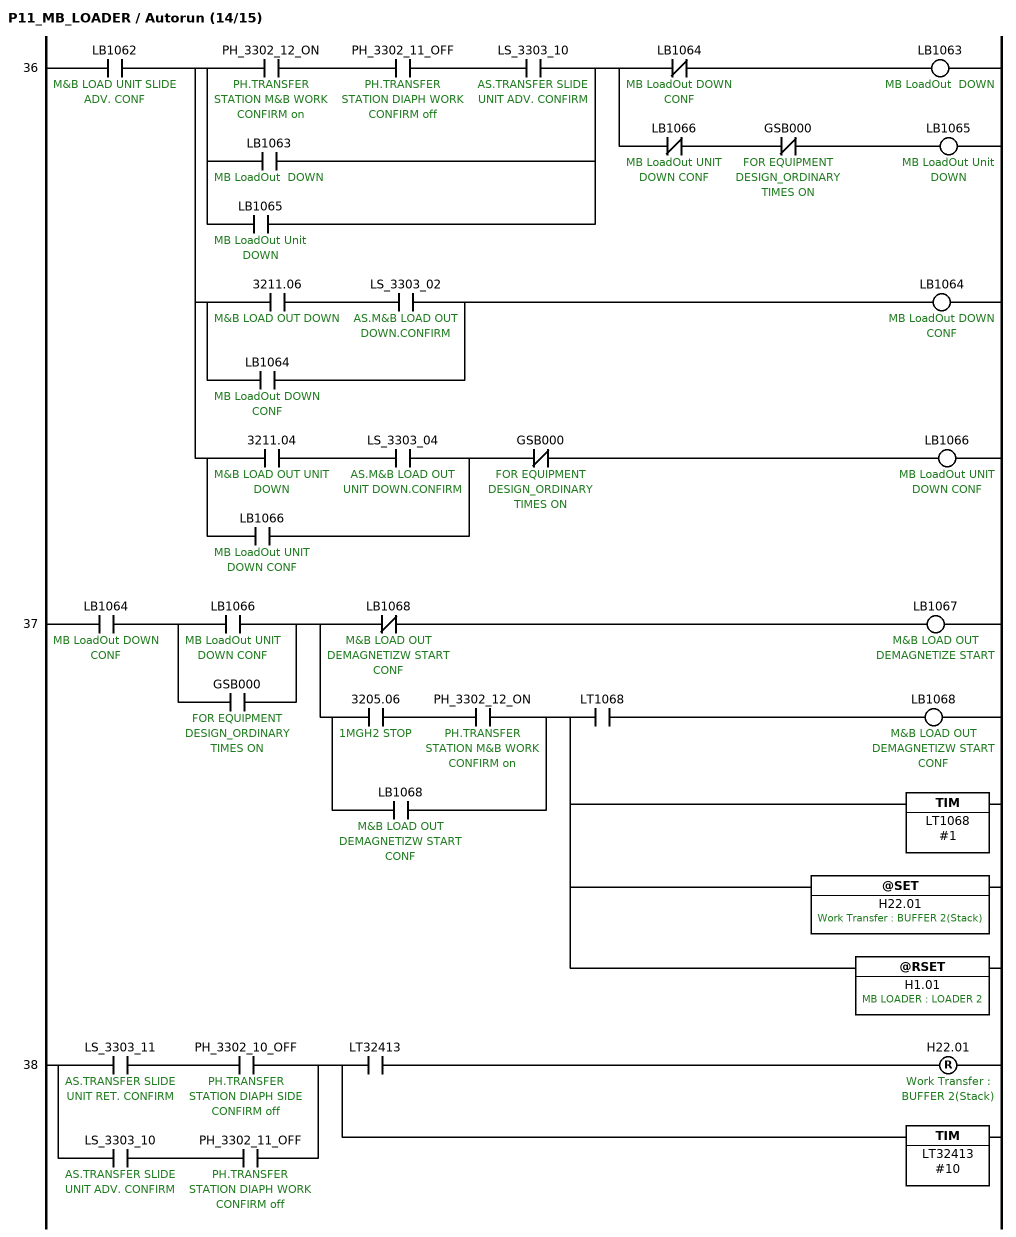
; rung 36
LD LB1062  ; M&B LOAD UNIT SLIDE ADV. CONF
OUT TR0
LD PH_3302_12_ON  ; PH.TRANSFER STATION M&B WORK CONFIRM on
AND PH_3302_11_OFF  ; PH.TRANSFER STATION DIAPH WORK CONFIRM off
AND LS_3303_10  ; AS.TRANSFER SLIDE UNIT ADV. CONFIRM
OR LB1063  ; MB LoadOut  DOWN
OR LB1065  ; MB LoadOut Unit  DOWN
ANDLD
OUT TR1
ANDNOT LB1064  ; MB LoadOut DOWN CONF
OUT LB1063  ; MB LoadOut  DOWN
LD TR1
ANDNOT LB1066  ; MB LoadOut UNIT DOWN CONF
ANDNOT GSB000  ; FOR EQUIPMENT DESIGN_ORDINARY TIMES ON
OUT LB1065  ; MB LoadOut Unit  DOWN
LD TR0
LD 3211.06  ; M&B LOAD OUT DOWN
AND LS_3303_02  ; AS.M&B LOAD OUT DOWN.CONFIRM
OR LB1064  ; MB LoadOut DOWN CONF
ANDLD
OUT LB1064  ; MB LoadOut DOWN CONF
LD TR0
LD 3211.04  ; M&B LOAD OUT UNIT DOWN
AND LS_3303_04  ; AS.M&B LOAD OUT UNIT DOWN.CONFIRM
OR LB1066  ; MB LoadOut UNIT DOWN CONF
ANDLD
ANDNOT GSB000  ; FOR EQUIPMENT DESIGN_ORDINARY TIMES ON
OUT LB1066  ; MB LoadOut UNIT DOWN CONF
; rung 37
LD LB1064  ; MB LoadOut DOWN CONF
LD LB1066  ; MB LoadOut UNIT DOWN CONF
OR GSB000  ; FOR EQUIPMENT DESIGN_ORDINARY TIMES ON
ANDLD
OUT TR0
ANDNOT LB1068  ; M&B LOAD OUT DEMAGNETIZW START CONF
OUT LB1067  ; M&B LOAD OUT DEMAGNETIZE START
LD TR0
LD 3205.06  ; 1MGH2 STOP
AND PH_3302_12_ON  ; PH.TRANSFER STATION M&B WORK CONFIRM on
OR LB1068  ; M&B LOAD OUT DEMAGNETIZW START CONF
ANDLD
OUT TR0
AND LT1068
OUT LB1068  ; M&B LOAD OUT DEMAGNETIZW START CONF
LD TR0
TIM LT1068 #1
@SET H22.01  ; Work Transfer : BUFFER 2(Stack)
@RSET H1.01  ; MB LOADER : LOADER 2
; rung 38
LD LS_3303_11  ; AS.TRANSFER SLIDE UNIT RET. CONFIRM
AND PH_3302_10_OFF  ; PH.TRANSFER STATION DIAPH SIDE CONFIRM off
LD LS_3303_10  ; AS.TRANSFER SLIDE UNIT ADV. CONFIRM
AND PH_3302_11_OFF  ; PH.TRANSFER STATION DIAPH WORK CONFIRM off
ORLD
OUT TR0
AND LT32413
RSET H22.01  ; Work Transfer : BUFFER 2(Stack)
LD TR0
TIM LT32413 #10

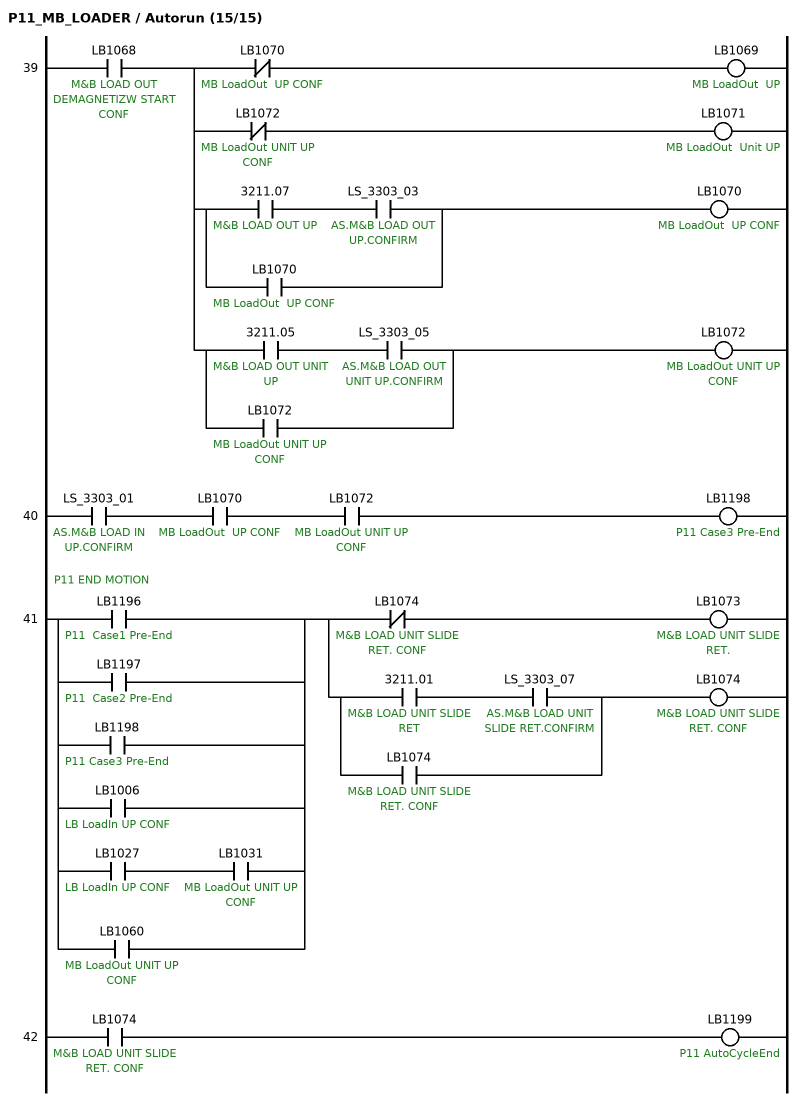
; rung 39
LD LB1068  ; M&B LOAD OUT DEMAGNETIZW START CONF
OUT TR0
ANDNOT LB1070  ; MB LoadOut  UP CONF
OUT LB1069  ; MB LoadOut  UP
LD TR0
ANDNOT LB1072  ; MB LoadOut UNIT UP CONF
OUT LB1071  ; MB LoadOut  Unit UP
LD TR0
LD 3211.07  ; M&B LOAD OUT UP
AND LS_3303_03  ; AS.M&B LOAD OUT UP.CONFIRM
OR LB1070  ; MB LoadOut  UP CONF
ANDLD
OUT LB1070  ; MB LoadOut  UP CONF
LD TR0
LD 3211.05  ; M&B LOAD OUT UNIT UP
AND LS_3303_05  ; AS.M&B LOAD OUT UNIT UP.CONFIRM
OR LB1072  ; MB LoadOut UNIT UP CONF
ANDLD
OUT LB1072  ; MB LoadOut UNIT UP CONF
; rung 40
LD LS_3303_01  ; AS.M&B LOAD IN UP.CONFIRM
AND LB1070  ; MB LoadOut  UP CONF
AND LB1072  ; MB LoadOut UNIT UP CONF
OUT LB1198  ; P11 Case3 Pre-End
; rung 41: P11 END MOTION
LD LB1196  ; P11  Case1 Pre-End
OR LB1197  ; P11  Case2 Pre-End
OR LB1198  ; P11 Case3 Pre-End
OR LB1006  ; LB LoadIn UP CONF
LD LB1027  ; LB LoadIn UP CONF
AND LB1031  ; MB LoadOut UNIT UP CONF
ORLD
OR LB1060  ; MB LoadOut UNIT UP CONF
OUT TR0
ANDNOT LB1074  ; M&B LOAD UNIT SLIDE RET. CONF
OUT LB1073  ; M&B LOAD UNIT SLIDE RET.
LD TR0
LD 3211.01  ; M&B LOAD UNIT SLIDE RET
AND LS_3303_07  ; AS.M&B LOAD UNIT SLIDE RET.CONFIRM
OR LB1074  ; M&B LOAD UNIT SLIDE RET. CONF
ANDLD
OUT LB1074  ; M&B LOAD UNIT SLIDE RET. CONF
; rung 42
LD LB1074  ; M&B LOAD UNIT SLIDE RET. CONF
OUT LB1199  ; P11 AutoCycleEnd

### Section Condition

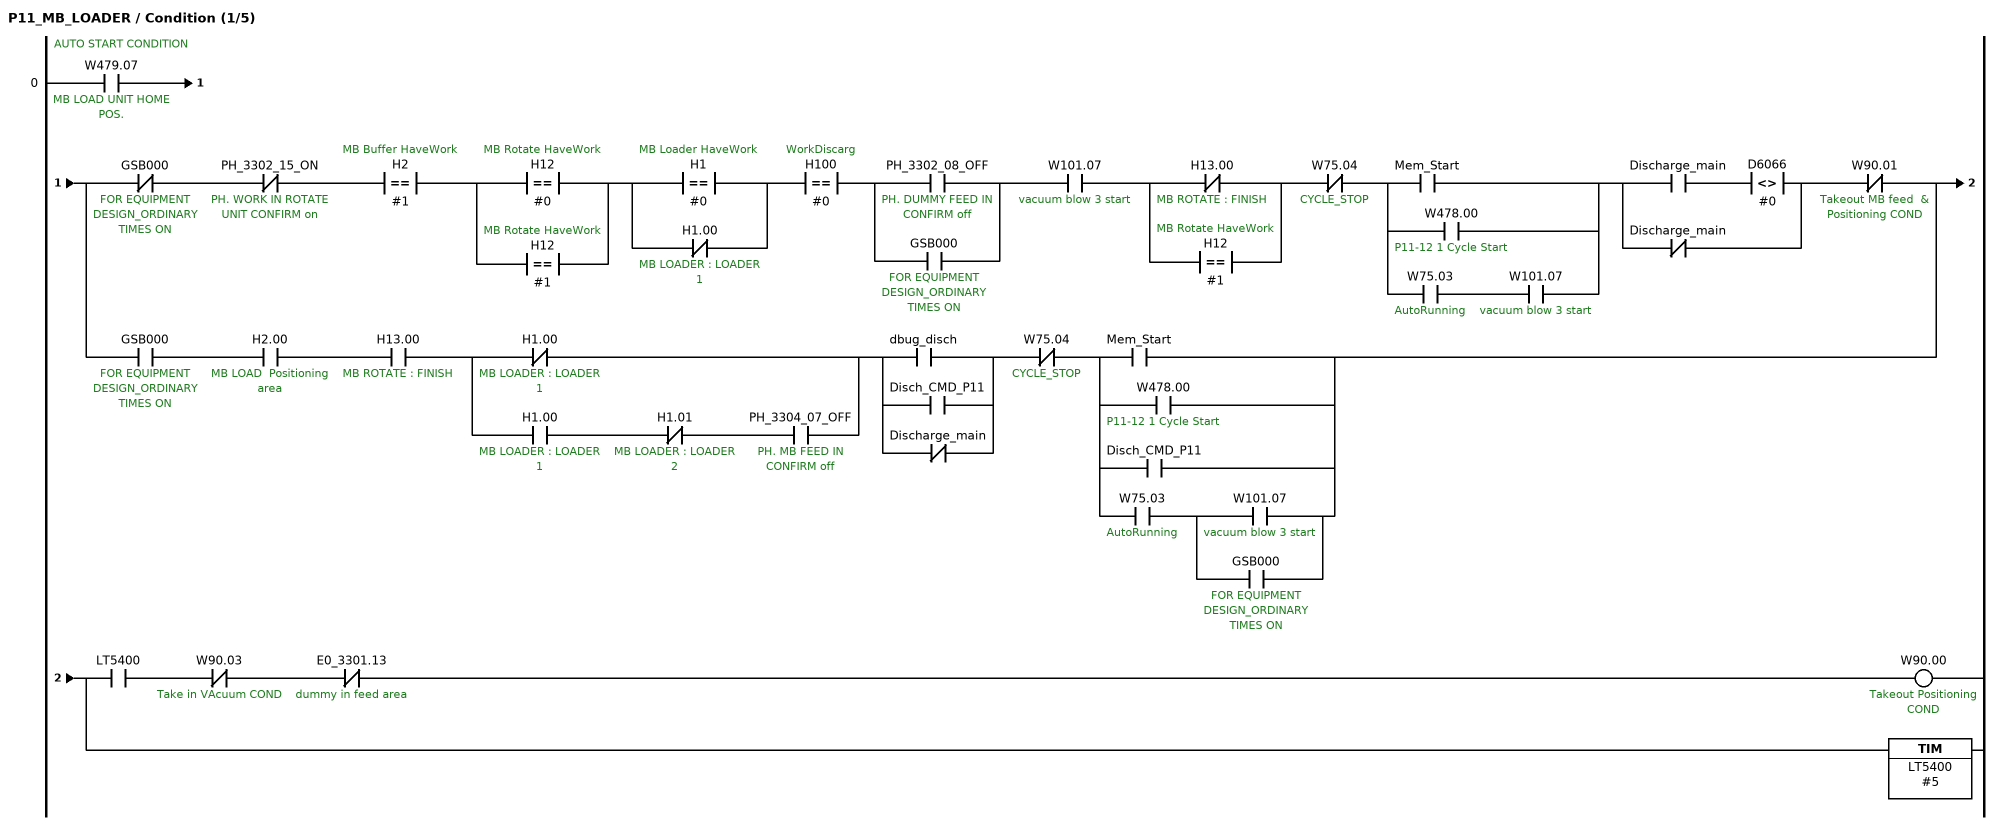
; rung 0: AUTO START CONDITION
LD W479.07  ; MB LOAD UNIT HOME POS.
LDNOT GSB000  ; FOR EQUIPMENT DESIGN_ORDINARY TIMES ON
ANDNOT PH_3302_15_ON  ; PH. WORK IN ROTATE UNIT CONFIRM on
AND=(300) H2 #1  ; MB Buffer HaveWork
LD=(300) H12 #0  ; MB Rotate HaveWork
OR=(300) H12 #1  ; MB Rotate HaveWork
ANDLD
LD=(300) H1 #0  ; MB Loader HaveWork
ORNOT H1.00  ; MB LOADER : LOADER 1
ANDLD
AND=(300) H100 #0  ; WorkDiscarg
LD PH_3302_08_OFF  ; PH. DUMMY FEED IN CONFIRM off
OR GSB000  ; FOR EQUIPMENT DESIGN_ORDINARY TIMES ON
ANDLD
AND W101.07  ; vacuum blow 3 start
LDNOT H13.00  ; MB ROTATE : FINISH
OR=(300) H12 #1  ; MB Rotate HaveWork
ANDLD
ANDNOT W75.04  ; CYCLE_STOP
LD Mem_Start
OR W478.00  ; P11-12 1 Cycle Start
LD W75.03  ; AutoRunning
AND W101.07  ; vacuum blow 3 start
ORLD
ANDLD
LD Discharge_main
AND<>(305) D6066 #0
ORNOT Discharge_main
ANDLD
ANDNOT W90.01  ; Takeout MB feed  & Positioning COND
LD GSB000  ; FOR EQUIPMENT DESIGN_ORDINARY TIMES ON
AND H2.00  ; MB LOAD  Positioning area
AND H13.00  ; MB ROTATE : FINISH
LDNOT H1.00  ; MB LOADER : LOADER 1
LD H1.00  ; MB LOADER : LOADER 1
ANDNOT H1.01  ; MB LOADER : LOADER 2
AND PH_3304_07_OFF  ; PH. MB FEED IN CONFIRM off
ORLD
ANDLD
LD dbug_disch
OR Disch_CMD_P11
ORNOT Discharge_main
ANDLD
ANDNOT W75.04  ; CYCLE_STOP
LD Mem_Start
OR W478.00  ; P11-12 1 Cycle Start
OR Disch_CMD_P11
LD W75.03  ; AutoRunning
LD W101.07  ; vacuum blow 3 start
OR GSB000  ; FOR EQUIPMENT DESIGN_ORDINARY TIMES ON
ANDLD
ORLD
ANDLD
ORLD
ANDLD
OUT TR0
AND LT5400
ANDNOT W90.03  ; Take in VAcuum COND
ANDNOT E0_3301.13  ; dummy in feed area
OUT W90.00  ; Takeout Positioning COND
LD TR0
TIM LT5400 #5

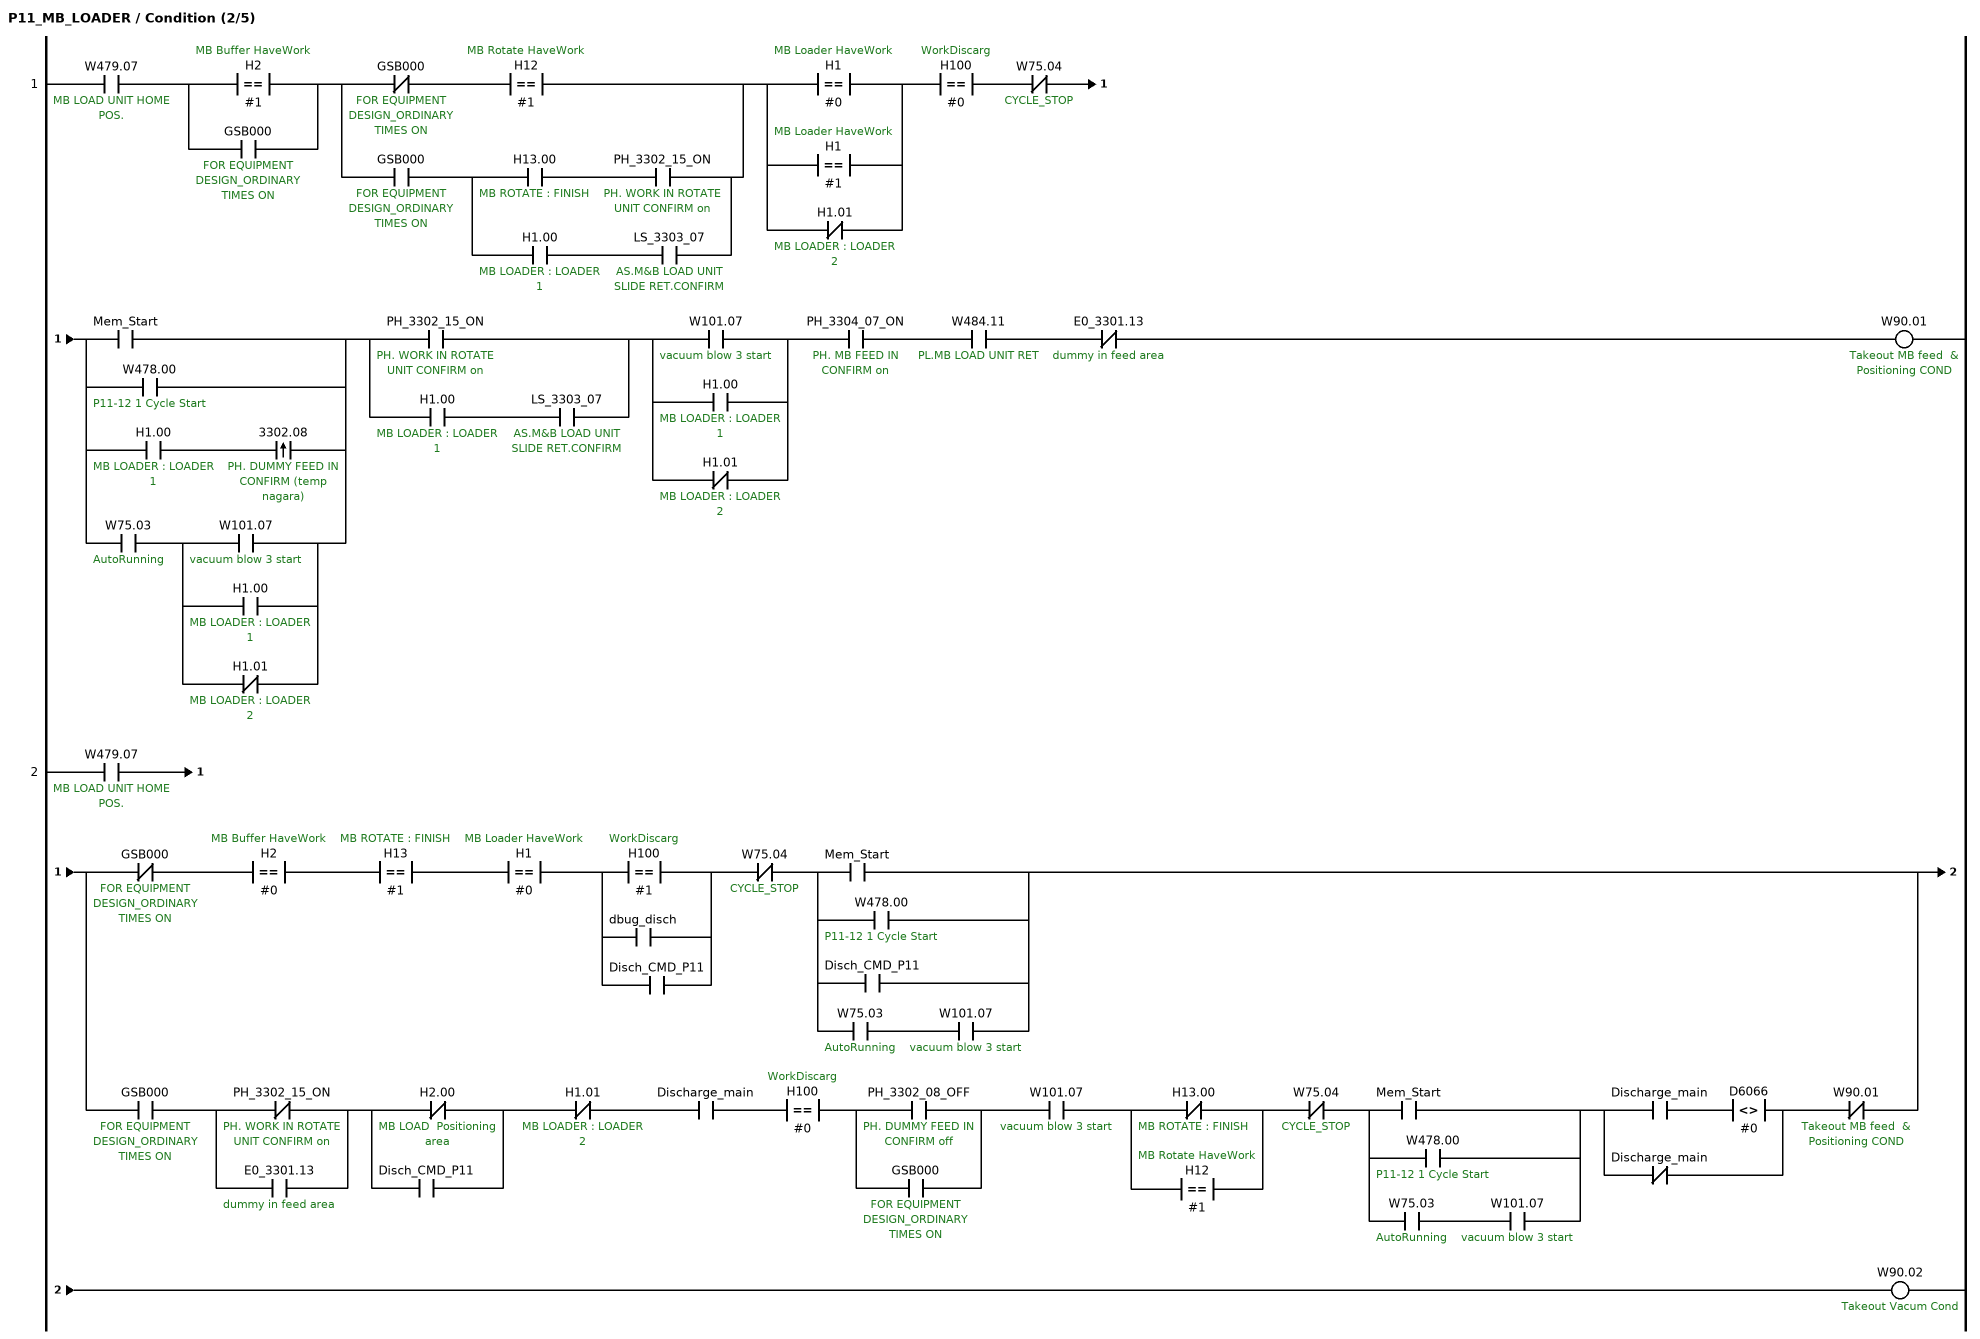
; rung 1
LD W479.07  ; MB LOAD UNIT HOME POS.
LD=(300) H2 #1  ; MB Buffer HaveWork
OR GSB000  ; FOR EQUIPMENT DESIGN_ORDINARY TIMES ON
ANDLD
LDNOT GSB000  ; FOR EQUIPMENT DESIGN_ORDINARY TIMES ON
AND=(300) H12 #1  ; MB Rotate HaveWork
LD GSB000  ; FOR EQUIPMENT DESIGN_ORDINARY TIMES ON
LD H13.00  ; MB ROTATE : FINISH
AND PH_3302_15_ON  ; PH. WORK IN ROTATE UNIT CONFIRM on
LD H1.00  ; MB LOADER : LOADER 1
AND LS_3303_07  ; AS.M&B LOAD UNIT SLIDE RET.CONFIRM
ORLD
ANDLD
ORLD
ANDLD
LD=(300) H1 #0  ; MB Loader HaveWork
OR=(300) H1 #1  ; MB Loader HaveWork
ORNOT H1.01  ; MB LOADER : LOADER 2
ANDLD
AND=(300) H100 #0  ; WorkDiscarg
ANDNOT W75.04  ; CYCLE_STOP
LD Mem_Start
OR W478.00  ; P11-12 1 Cycle Start
LD H1.00  ; MB LOADER : LOADER 1
@AND 3302.08  ; PH. DUMMY FEED IN CONFIRM (temp nagara)
ORLD
LD W75.03  ; AutoRunning
LD W101.07  ; vacuum blow 3 start
OR H1.00  ; MB LOADER : LOADER 1
ORNOT H1.01  ; MB LOADER : LOADER 2
ANDLD
ORLD
ANDLD
LD PH_3302_15_ON  ; PH. WORK IN ROTATE UNIT CONFIRM on
LD H1.00  ; MB LOADER : LOADER 1
AND LS_3303_07  ; AS.M&B LOAD UNIT SLIDE RET.CONFIRM
ORLD
ANDLD
LD W101.07  ; vacuum blow 3 start
OR H1.00  ; MB LOADER : LOADER 1
ORNOT H1.01  ; MB LOADER : LOADER 2
ANDLD
AND PH_3304_07_ON  ; PH. MB FEED IN CONFIRM on
AND W484.11  ; PL.MB LOAD UNIT RET
ANDNOT E0_3301.13  ; dummy in feed area
OUT W90.01  ; Takeout MB feed  & Positioning COND
; rung 2
LD W479.07  ; MB LOAD UNIT HOME POS.
LDNOT GSB000  ; FOR EQUIPMENT DESIGN_ORDINARY TIMES ON
AND=(300) H2 #0  ; MB Buffer HaveWork
AND=(300) H13 #1  ; MB ROTATE : FINISH
AND=(300) H1 #0  ; MB Loader HaveWork
LD=(300) H100 #1  ; WorkDiscarg
OR dbug_disch
OR Disch_CMD_P11
ANDLD
ANDNOT W75.04  ; CYCLE_STOP
LD Mem_Start
OR W478.00  ; P11-12 1 Cycle Start
OR Disch_CMD_P11
LD W75.03  ; AutoRunning
AND W101.07  ; vacuum blow 3 start
ORLD
ANDLD
LD GSB000  ; FOR EQUIPMENT DESIGN_ORDINARY TIMES ON
LDNOT PH_3302_15_ON  ; PH. WORK IN ROTATE UNIT CONFIRM on
OR E0_3301.13  ; dummy in feed area
ANDLD
LDNOT H2.00  ; MB LOAD  Positioning area
OR Disch_CMD_P11
ANDLD
ANDNOT H1.01  ; MB LOADER : LOADER 2
AND Discharge_main
AND=(300) H100 #0  ; WorkDiscarg
LD PH_3302_08_OFF  ; PH. DUMMY FEED IN CONFIRM off
OR GSB000  ; FOR EQUIPMENT DESIGN_ORDINARY TIMES ON
ANDLD
AND W101.07  ; vacuum blow 3 start
LDNOT H13.00  ; MB ROTATE : FINISH
OR=(300) H12 #1  ; MB Rotate HaveWork
ANDLD
ANDNOT W75.04  ; CYCLE_STOP
LD Mem_Start
OR W478.00  ; P11-12 1 Cycle Start
LD W75.03  ; AutoRunning
AND W101.07  ; vacuum blow 3 start
ORLD
ANDLD
LD Discharge_main
AND<>(305) D6066 #0
ORNOT Discharge_main
ANDLD
ANDNOT W90.01  ; Takeout MB feed  & Positioning COND
ORLD
ANDLD
OUT W90.02  ; Takeout Vacum Cond

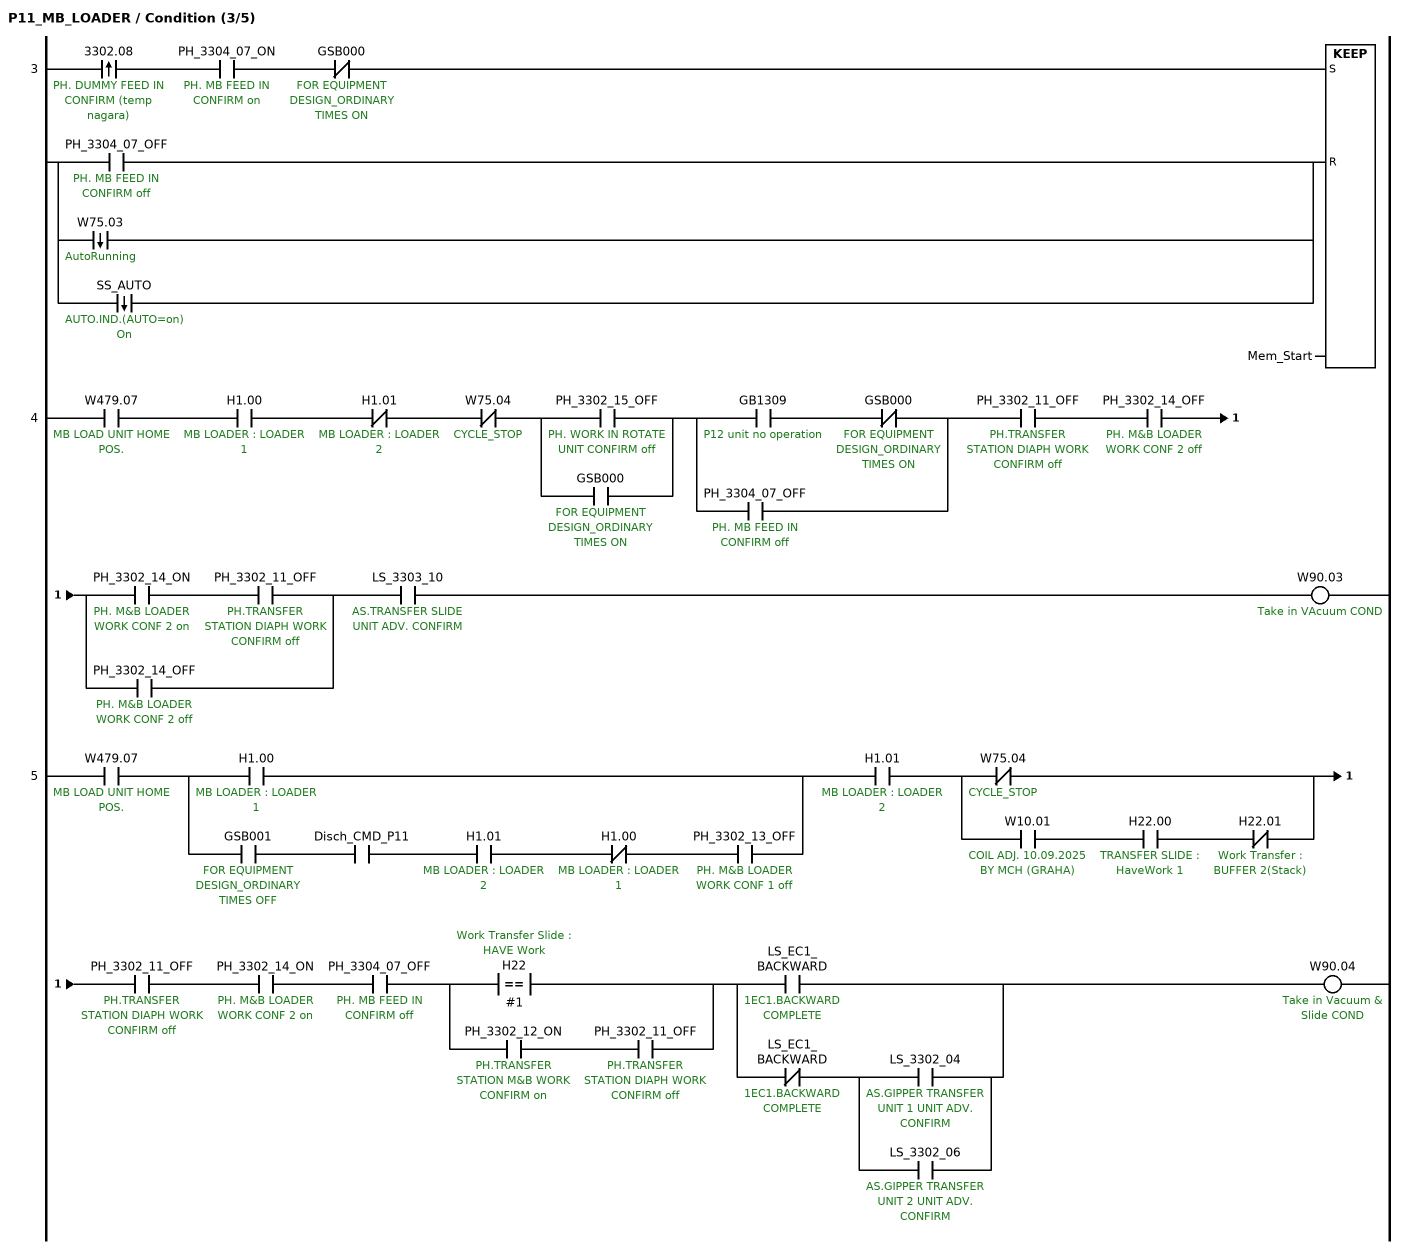
; rung 3
@LD 3302.08  ; PH. DUMMY FEED IN CONFIRM (temp nagara)
AND PH_3304_07_ON  ; PH. MB FEED IN CONFIRM on
ANDNOT GSB000  ; FOR EQUIPMENT DESIGN_ORDINARY TIMES ON
LD PH_3304_07_OFF  ; PH. MB FEED IN CONFIRM off
%OR W75.03  ; AutoRunning
%OR SS_AUTO  ; AUTO.IND.(AUTO=on) On
KEEP Mem_Start
; rung 4
LD W479.07  ; MB LOAD UNIT HOME POS.
AND H1.00  ; MB LOADER : LOADER 1
ANDNOT H1.01  ; MB LOADER : LOADER 2
ANDNOT W75.04  ; CYCLE_STOP
LD PH_3302_15_OFF  ; PH. WORK IN ROTATE UNIT CONFIRM off
OR GSB000  ; FOR EQUIPMENT DESIGN_ORDINARY TIMES ON
ANDLD
LD GB1309  ; P12 unit no operation
ANDNOT GSB000  ; FOR EQUIPMENT DESIGN_ORDINARY TIMES ON
OR PH_3304_07_OFF  ; PH. MB FEED IN CONFIRM off
ANDLD
AND PH_3302_11_OFF  ; PH.TRANSFER STATION DIAPH WORK CONFIRM off
AND PH_3302_14_OFF  ; PH. M&B LOADER WORK CONF 2 off
LD PH_3302_14_ON  ; PH. M&B LOADER WORK CONF 2 on
AND PH_3302_11_OFF  ; PH.TRANSFER STATION DIAPH WORK CONFIRM off
OR PH_3302_14_OFF  ; PH. M&B LOADER WORK CONF 2 off
ANDLD
AND LS_3303_10  ; AS.TRANSFER SLIDE UNIT ADV. CONFIRM
OUT W90.03  ; Take in VAcuum COND
; rung 5
LD W479.07  ; MB LOAD UNIT HOME POS.
LD H1.00  ; MB LOADER : LOADER 1
LD GSB001  ; FOR EQUIPMENT DESIGN_ORDINARY TIMES OFF
AND Disch_CMD_P11
AND H1.01  ; MB LOADER : LOADER 2
ANDNOT H1.00  ; MB LOADER : LOADER 1
AND PH_3302_13_OFF  ; PH. M&B LOADER WORK CONF 1 off
ORLD
ANDLD
AND H1.01  ; MB LOADER : LOADER 2
LDNOT W75.04  ; CYCLE_STOP
LD W10.01  ; COIL ADJ. 10.09.2025 BY MCH (GRAHA)
AND H22.00  ; TRANSFER SLIDE : HaveWork 1
ANDNOT H22.01  ; Work Transfer : BUFFER 2(Stack)
ORLD
ANDLD
AND PH_3302_11_OFF  ; PH.TRANSFER STATION DIAPH WORK CONFIRM off
AND PH_3302_14_ON  ; PH. M&B LOADER WORK CONF 2 on
AND PH_3304_07_OFF  ; PH. MB FEED IN CONFIRM off
LD=(300) H22 #1  ; Work Transfer Slide : HAVE Work
LD PH_3302_12_ON  ; PH.TRANSFER STATION M&B WORK CONFIRM on
AND PH_3302_11_OFF  ; PH.TRANSFER STATION DIAPH WORK CONFIRM off
ORLD
ANDLD
LD LS_EC1_BACKWARD  ; 1EC1.BACKWARD COMPLETE
LDNOT LS_EC1_BACKWARD  ; 1EC1.BACKWARD COMPLETE
LD LS_3302_04  ; AS.GIPPER TRANSFER UNIT 1 UNIT ADV. CONFIRM
OR LS_3302_06  ; AS.GIPPER TRANSFER UNIT 2 UNIT ADV. CONFIRM
ANDLD
ORLD
ANDLD
OUT W90.04  ; Take in Vacuum & Slide COND

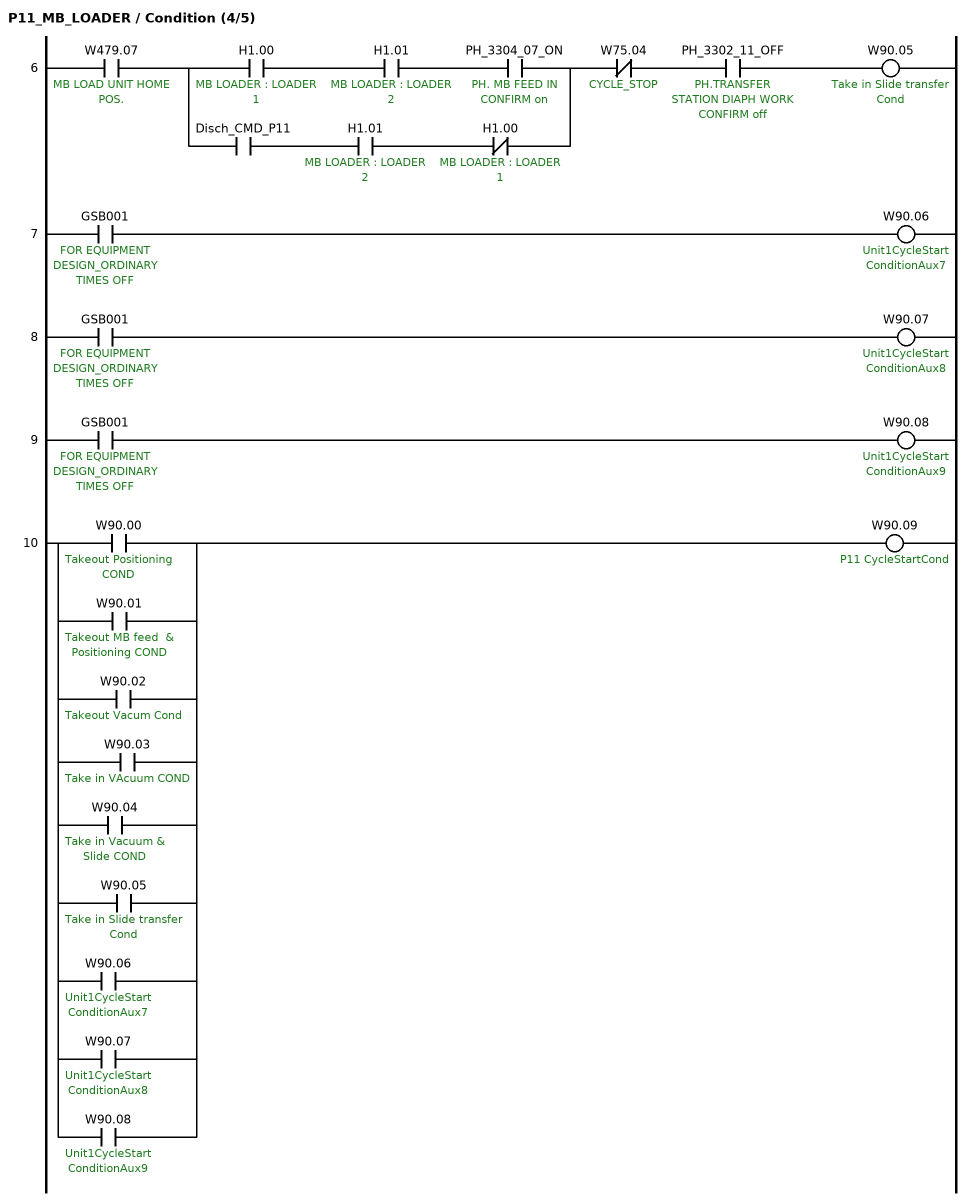
; rung 6
LD W479.07  ; MB LOAD UNIT HOME POS.
LD H1.00  ; MB LOADER : LOADER 1
AND H1.01  ; MB LOADER : LOADER 2
AND PH_3304_07_ON  ; PH. MB FEED IN CONFIRM on
LD Disch_CMD_P11
AND H1.01  ; MB LOADER : LOADER 2
ANDNOT H1.00  ; MB LOADER : LOADER 1
ORLD
ANDLD
ANDNOT W75.04  ; CYCLE_STOP
AND PH_3302_11_OFF  ; PH.TRANSFER STATION DIAPH WORK CONFIRM off
OUT W90.05  ; Take in Slide transfer Cond
; rung 7
LD GSB001  ; FOR EQUIPMENT DESIGN_ORDINARY TIMES OFF
OUT W90.06  ; Unit1CycleStartConditionAux7
; rung 8
LD GSB001  ; FOR EQUIPMENT DESIGN_ORDINARY TIMES OFF
OUT W90.07  ; Unit1CycleStartConditionAux8
; rung 9
LD GSB001  ; FOR EQUIPMENT DESIGN_ORDINARY TIMES OFF
OUT W90.08  ; Unit1CycleStartConditionAux9
; rung 10
LD W90.00  ; Takeout Positioning COND
OR W90.01  ; Takeout MB feed  & Positioning COND
OR W90.02  ; Takeout Vacum Cond
OR W90.03  ; Take in VAcuum COND
OR W90.04  ; Take in Vacuum & Slide COND
OR W90.05  ; Take in Slide transfer Cond
OR W90.06  ; Unit1CycleStartConditionAux7
OR W90.07  ; Unit1CycleStartConditionAux8
OR W90.08  ; Unit1CycleStartConditionAux9
OUT W90.09  ; P11 CycleStartCond

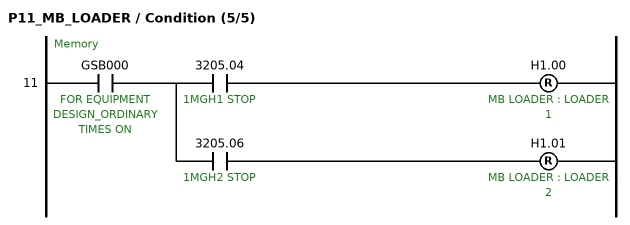
; rung 11: Memory
LD GSB000  ; FOR EQUIPMENT DESIGN_ORDINARY TIMES ON
OUT TR0
AND 3205.04  ; 1MGH1 STOP
RSET H1.00  ; MB LOADER : LOADER 1
LD TR0
AND 3205.06  ; 1MGH2 STOP
RSET H1.01  ; MB LOADER : LOADER 2

### Section Device_Output

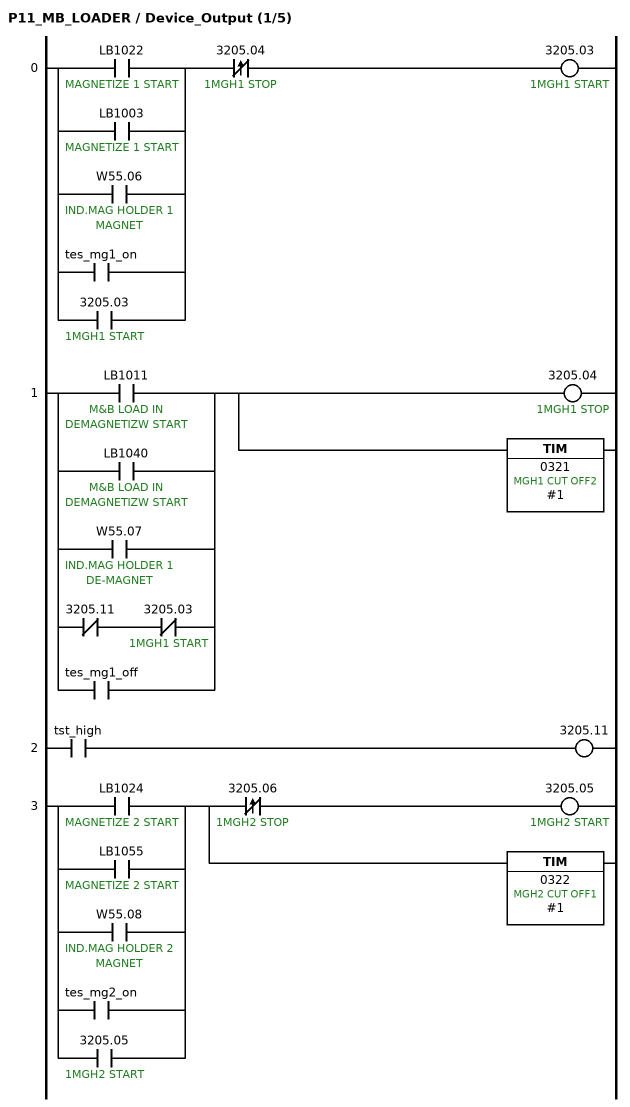
; rung 0
LD LB1022  ; MAGNETIZE 1 START
OR LB1003  ; MAGNETIZE 1 START
OR W55.06  ; IND.MAG HOLDER 1 MAGNET
OR tes_mg1_on
OR 3205.03  ; 1MGH1 START
@ANDNOT 3205.04  ; 1MGH1 STOP
OUT 3205.03  ; 1MGH1 START
; rung 1
LD LB1011  ; M&B LOAD IN DEMAGNETIZW START
OR LB1040  ; M&B LOAD IN DEMAGNETIZW START
OR W55.07  ; IND.MAG HOLDER 1 DE-MAGNET
LDNOT 3205.11
ANDNOT 3205.03  ; 1MGH1 START
ORLD
OR tes_mg1_off
OUT 3205.04  ; 1MGH1 STOP
TIM 0321 #1  ; MGH1 CUT OFF2
; rung 2
LD tst_high
OUT 3205.11
; rung 3
LD LB1024  ; MAGNETIZE 2 START
OR LB1055  ; MAGNETIZE 2 START
OR W55.08  ; IND.MAG HOLDER 2 MAGNET
OR tes_mg2_on
OR 3205.05  ; 1MGH2 START
OUT TR0
@ANDNOT 3205.06  ; 1MGH2 STOP
OUT 3205.05  ; 1MGH2 START
LD TR0
TIM 0322 #1  ; MGH2 CUT OFF1

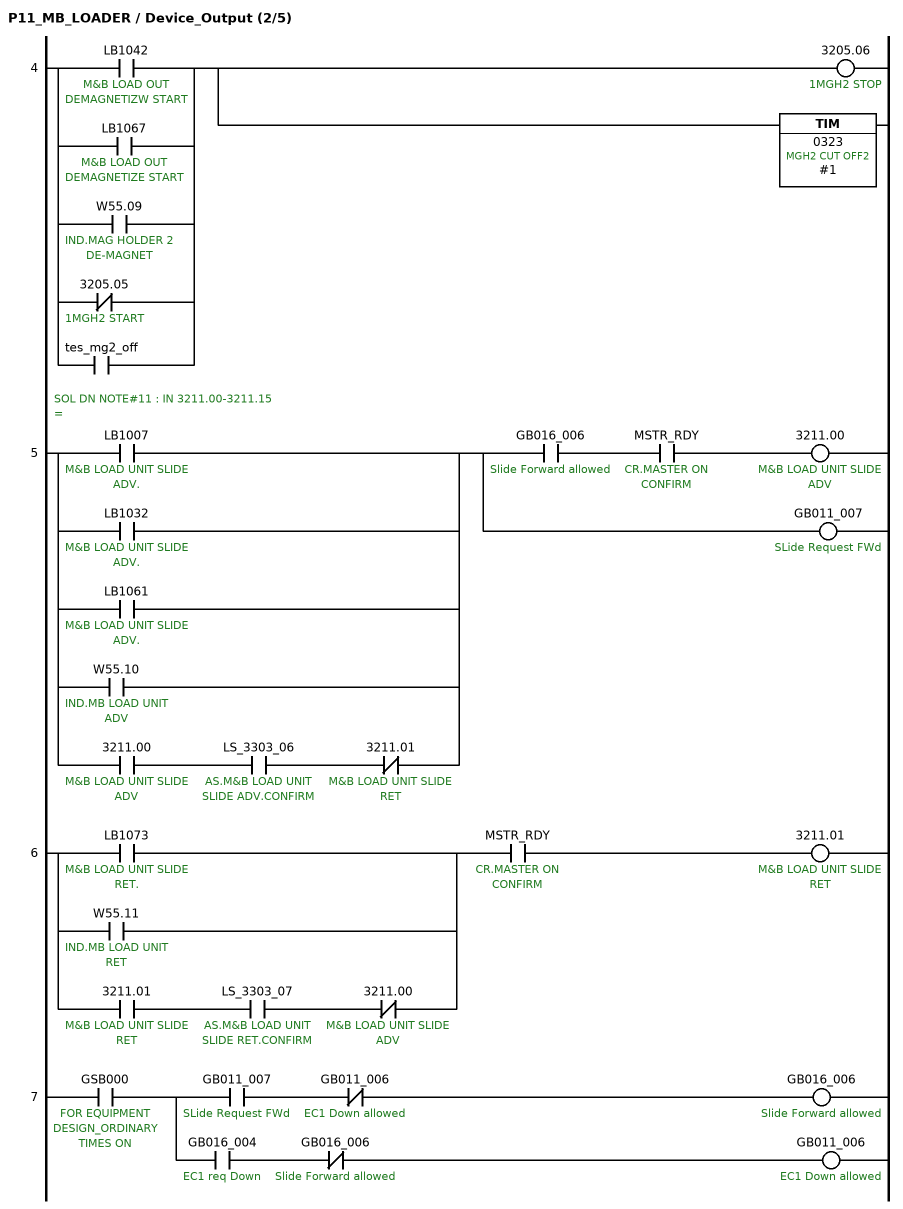
; rung 4
LD LB1042  ; M&B LOAD OUT DEMAGNETIZW START
OR LB1067  ; M&B LOAD OUT DEMAGNETIZE START
OR W55.09  ; IND.MAG HOLDER 2 DE-MAGNET
ORNOT 3205.05  ; 1MGH2 START
OR tes_mg2_off
OUT 3205.06  ; 1MGH2 STOP
TIM 0323 #1  ; MGH2 CUT OFF2
; rung 5: SOL DN NOTE#11 : IN 3211.00-3211.15 / =
LD LB1007  ; M&B LOAD UNIT SLIDE ADV.
OR LB1032  ; M&B LOAD UNIT SLIDE ADV.
OR LB1061  ; M&B LOAD UNIT SLIDE ADV.
OR W55.10  ; IND.MB LOAD UNIT ADV
LD 3211.00  ; M&B LOAD UNIT SLIDE ADV
AND LS_3303_06  ; AS.M&B LOAD UNIT SLIDE ADV.CONFIRM
ANDNOT 3211.01  ; M&B LOAD UNIT SLIDE RET
ORLD
OUT TR0
AND GB016_006  ; Slide Forward allowed
AND MSTR_RDY  ; CR.MASTER ON CONFIRM
OUT 3211.00  ; M&B LOAD UNIT SLIDE ADV
LD TR0
OUT GB011_007  ; SLide Request FWd
; rung 6
LD LB1073  ; M&B LOAD UNIT SLIDE RET.
OR W55.11  ; IND.MB LOAD UNIT RET
LD 3211.01  ; M&B LOAD UNIT SLIDE RET
AND LS_3303_07  ; AS.M&B LOAD UNIT SLIDE RET.CONFIRM
ANDNOT 3211.00  ; M&B LOAD UNIT SLIDE ADV
ORLD
AND MSTR_RDY  ; CR.MASTER ON CONFIRM
OUT 3211.01  ; M&B LOAD UNIT SLIDE RET
; rung 7
LD GSB000  ; FOR EQUIPMENT DESIGN_ORDINARY TIMES ON
OUT TR0
AND GB011_007  ; SLide Request FWd
ANDNOT GB011_006  ; EC1 Down allowed
OUT GB016_006  ; Slide Forward allowed
LD TR0
AND GB016_004  ; EC1 req Down
ANDNOT GB016_006  ; Slide Forward allowed
OUT GB011_006  ; EC1 Down allowed

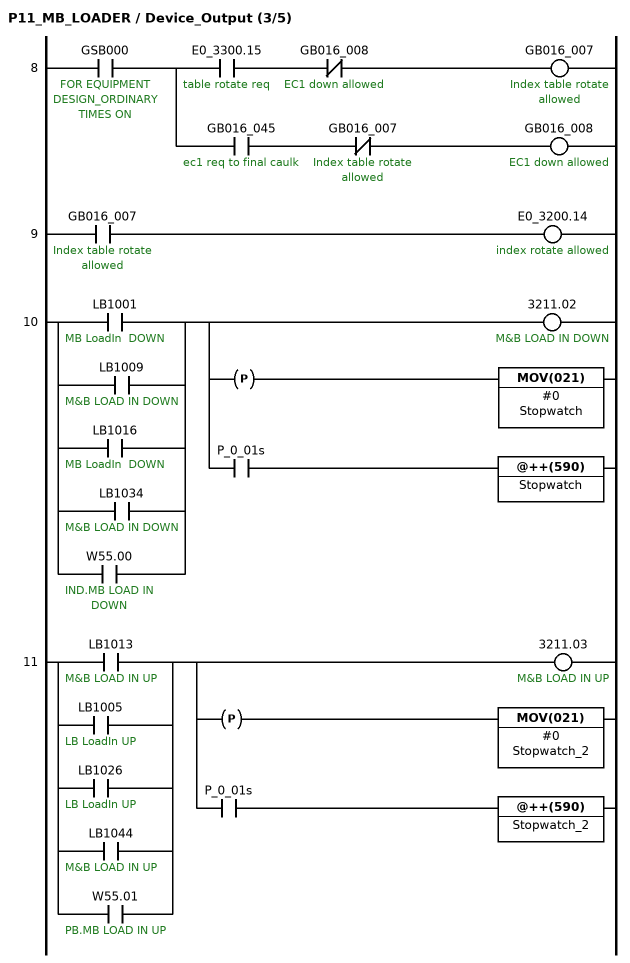
; rung 8
LD GSB000  ; FOR EQUIPMENT DESIGN_ORDINARY TIMES ON
OUT TR0
AND E0_3300.15  ; table rotate req
ANDNOT GB016_008  ; EC1 down allowed
OUT GB016_007  ; Index table rotate allowed
LD TR0
AND GB016_045  ; ec1 req to final caulk
ANDNOT GB016_007  ; Index table rotate allowed
OUT GB016_008  ; EC1 down allowed
; rung 9
LD GB016_007  ; Index table rotate allowed
OUT E0_3200.14  ; index rotate allowed
; rung 10
LD LB1001  ; MB LoadIn  DOWN
OR LB1009  ; M&B LOAD IN DOWN
OR LB1016  ; MB LoadIn  DOWN
OR LB1034  ; M&B LOAD IN DOWN
OR W55.00  ; IND.MB LOAD IN DOWN
OUT TR0
OUT 3211.02  ; M&B LOAD IN DOWN
UP(521)
MOV(021) #0 Stopwatch
LD TR0
AND P_0_01s
@++(590) Stopwatch
; rung 11
LD LB1013  ; M&B LOAD IN UP
OR LB1005  ; LB LoadIn UP
OR LB1026  ; LB LoadIn UP
OR LB1044  ; M&B LOAD IN UP
OR W55.01  ; PB.MB LOAD IN UP
OUT TR0
OUT 3211.03  ; M&B LOAD IN UP
UP(521)
MOV(021) #0 Stopwatch_2
LD TR0
AND P_0_01s
@++(590) Stopwatch_2

